LIN {X 0,Y 573.233,Z 312.707,A -85,B 0,C 180,E1 -2302.192,E2 -2302.192} C_VEL
LIN {X 0,Y 573.235,Z 312.7,A -85,B 0,C 180,E1 -2305.229,E2 -2305.229} C_VEL
LIN {X 0,Y 573.253,Z 312.699,A -85,B 0,C 180,E1 -2307.772,E2 -2307.772} C_VEL
LIN {X 0,Y 573.264,Z 312.7,A -85,B 0,C 180,E1 -2310.634,E2 -2310.634} C_VEL
LIN {X 0,Y 573.212,Z 312.703,A -85,B 0,C 180,E1 -2313.514,E2 -2313.514} C_VEL
LIN {X 0,Y 573.23,Z 312.71,A -85,B 0,C 180,E1 -2316.135,E2 -2316.135} C_VEL
LIN {X 0,Y 573.252,Z 312.697,A -85,B 0,C 180,E1 -2319.174,E2 -2319.174} C_VEL
LIN {X 0,Y 573.218,Z 312.702,A -85,B 0,C 180,E1 -2321.411,E2 -2321.411} C_VEL
LIN {X 0,Y 573.244,Z 312.701,A -85,B 0,C 180,E1 -2323.622,E2 -2323.622} C_VEL
LIN {X 0,Y 573.276,Z 312.7,A -85,B 0,C 180,E1 -2325.807,E2 -2325.807} C_VEL
LIN {X 0,Y 573.268,Z 312.696,A -85,B 0,C 180,E1 -2328.745,E2 -2328.745} C_VEL
LIN {X 0,Y 573.254,Z 312.7,A -85,B 0,C 180,E1 -2331.54,E2 -2331.54} C_VEL
LIN {X 0,Y 573.274,Z 312.698,A -85,B 0,C 180,E1 -2334.372,E2 -2334.372} C_VEL
LIN {X 0,Y 573.308,Z 312.699,A -85,B 0,C 180,E1 -2337.893,E2 -2337.893} C_VEL
LIN {X 0,Y 573.318,Z 312.697,A -85,B 0,C 180,E1 -2340,E2 -2340} C_VEL
LIN {X 0,Y 573.287,Z 312.693,A -85,B 0,C 180,E1 -2342.811,E2 -2342.811} C_VEL
LIN {X 0,Y 573.28,Z 312.701,A -85,B 0,C 180,E1 -2345.629,E2 -2345.629} C_VEL
LIN {X 0,Y 573.239,Z 312.7,A -85,B 0,C 180,E1 -2348.46,E2 -2348.46} C_VEL
LIN {X 0,Y 573.277,Z 312.697,A -85,B 0,C 180,E1 -2351.312,E2 -2351.312} C_VEL
LIN {X 0,Y 573.262,Z 312.697,A -85,B 0,C 180,E1 -2354.415,E2 -2354.415} C_VEL
LIN {X 0,Y 573.181,Z 312.707,A -85,B 0,C 180,E1 -2357.114,E2 -2357.114} C_VEL
LIN {X 0,Y 573.27,Z 312.7,A -85,B 0,C 180,E1 -2359.33,E2 -2359.33} C_VEL
LIN {X 0,Y 573.199,Z 312.705,A -85,B 0,C 180,E1 -2362.34,E2 -2362.34} C_VEL
LIN {X 0,Y 573.197,Z 312.704,A -85,B 0,C 180,E1 -2364.342,E2 -2364.342} C_VEL
LIN {X 0,Y 572.56,Z 312.785,A -85,B 0,C 180,E1 -2364.928,E2 -2364.928} C_VEL
LIN {X 0,Y 569.728,Z 313.143,A -85,B 0,C 180,E1 -2365.88,E2 -2365.88} C_VEL
LIN {X 0,Y 567.308,Z 313.449,A -85,B 0,C 180,E1 -2366.645,E2 -2366.645} C_VEL
LIN {X 0,Y 566.25,Z 313.578,A -85,B 0,C 180,E1 -2367.236,E2 -2367.236} C_VEL
LIN {X 0,Y 566.155,Z 313.587,A -85,B 0,C 180,E1 -2367.437,E2 -2367.437} C_VEL
LIN {X 0,Y 566.151,Z 313.584,A -85,B 0,C 180,E1 -2369.772,E2 -2369.772} C_VEL
LIN {X 0,Y 566.181,Z 313.578,A -85,B 0,C 180,E1 -2372.425,E2 -2372.425} C_VEL
LIN {X 0,Y 566.162,Z 313.584,A -85,B 0,C 180,E1 -2374.986,E2 -2374.986} C_VEL
LIN {X 0,Y 566.18,Z 313.586,A -85,B 0,C 180,E1 -2377.463,E2 -2377.463} C_VEL
LIN {X 0,Y 566.159,Z 313.581,A -85,B 0,C 180,E1 -2380.204,E2 -2380.204} C_VEL
LIN {X 0,Y 566.145,Z 313.589,A -85,B 0,C 180,E1 -2383.06,E2 -2383.06} C_VEL
LIN {X 0,Y 566.136,Z 313.584,A -85,B 0,C 180,E1 -2386.056,E2 -2386.056} C_VEL
LIN {X 0,Y 566.124,Z 313.59,A -85,B 0,C 180,E1 -2388.856,E2 -2388.856} C_VEL
LIN {X 0,Y 566.157,Z 313.589,A -85,B 0,C 180,E1 -2391.449,E2 -2391.449} C_VEL
LIN {X 0,Y 566.135,Z 313.585,A -85,B 0,C 180,E1 -2394.306,E2 -2394.306} C_VEL
LIN {X 0,Y 566.154,Z 313.588,A -85,B 0,C 180,E1 -2396.893,E2 -2396.893} C_VEL
LIN {X 0,Y 566.151,Z 313.59,A -85,B 0,C 180,E1 -2399.405,E2 -2399.405} C_VEL
LIN {X 0,Y 566.145,Z 313.587,A -85,B 0,C 180,E1 -2401.854,E2 -2401.854} C_VEL
LIN {X 0,Y 566.187,Z 313.691,A -85,B 0,C 180,E1 -2403.507,E2 -2403.507} C_VEL
LIN {X 0,Y 566.832,Z 319.406,A -85,B 0,C 180,E1 -2404.447,E2 -2404.447} C_VEL
LIN {X 0,Y 566.58,Z 337.004,A -85,B 0,C 180,E1 -2407.193,E2 -2407.193} C_VEL
LIN {X 0,Y 566.557,Z 342.716,A -85,B 0,C 180,E1 -2408.077,E2 -2408.077} C_VEL
LIN {X 0,Y 567.74,Z 348.996,A -85,B 0,C 180,E1 -2408.2,E2 -2408.2} C_VEL
LIN {X 0,Y 567.437,Z 479.381,A -85,B 0,C 180,E1 -2409.89,E2 -2409.89} C_VEL
LIN {X 0,Y 567.328,Z 493.858,A -85,B 0,C 180,E1 -2410.226,E2 -2410.226} C_VEL
LIN {X 0,Y 567.16,Z 507.522,A -85,B 0,C 180,E1 -2410.689,E2 -2410.689} C_VEL
LIN {X 0,Y 567.009,Z 520.891,A -85,B 0,C 180,E1 -2411.294,E2 -2411.294} C_VEL
LIN {X 0,Y 566.777,Z 533.749,A -85,B 0,C 180,E1 -2412.034,E2 -2412.034} C_VEL
LIN {X 0,Y 566.592,Z 545.641,A -85,B 0,C 180,E1 -2412.884,E2 -2412.884} C_VEL
LIN {X 0,Y 566.402,Z 556.077,A -85,B 0,C 180,E1 -2413.788,E2 -2413.788} C_VEL
LIN {X 0,Y 566.259,Z 566.633,A -85,B 0,C 180,E1 -2414.892,E2 -2414.892} C_VEL
LIN {X 0,Y 566.111,Z 575.295,A -85,B 0,C 180,E1 -2415.99,E2 -2415.99} C_VEL
LIN {X 0,Y 566.022,Z 583.527,A -85,B 0,C 180,E1 -2417.268,E2 -2417.268} C_VEL
LIN {X 0,Y 565.938,Z 590.127,A -85,B 0,C 180,E1 -2418.539,E2 -2418.539} C_VEL
LIN {X 0,Y 565.917,Z 594.689,A -85,B 0,C 180,E1 -2419.626,E2 -2419.626} C_VEL
LIN {X 0,Y 565.877,Z 598.259,A -85,B 0,C 180,E1 -2420.709,E2 -2420.709} C_VEL
LIN {X 0,Y 565.882,Z 601.734,A -85,B 0,C 180,E1 -2422.148,E2 -2422.148} C_VEL
LIN {X 0,Y 565.899,Z 603.791,A -85,B 0,C 180,E1 -2423.582,E2 -2423.582} C_VEL
LIN {X 0,Y 565.843,Z 604.498,A -85,B 0,C 180,E1 -2425.012,E2 -2425.012} C_VEL
LIN {X 0,Y 565.885,Z 603.864,A -85,B 0,C 180,E1 -2426.44,E2 -2426.44} C_VEL
LIN {X 0,Y 565.839,Z 601.889,A -85,B 0,C 180,E1 -2427.865,E2 -2427.865} C_VEL
LIN {X 0,Y 565.848,Z 598.534,A -85,B 0,C 180,E1 -2429.288,E2 -2429.288} C_VEL
LIN {X 0,Y 565.89,Z 593.71,A -85,B 0,C 180,E1 -2430.712,E2 -2430.712} C_VEL
LIN {X 0,Y 566.002,Z 589.069,A -85,B 0,C 180,E1 -2431.779,E2 -2431.779} C_VEL
LIN {X 0,Y 566.061,Z 582.343,A -85,B 0,C 180,E1 -2433.025,E2 -2433.025} C_VEL
LIN {X 0,Y 566.16,Z 574.011,A -85,B 0,C 180,E1 -2434.271,E2 -2434.271} C_VEL
LIN {X 0,Y 566.241,Z 565.352,A -85,B 0,C 180,E1 -2435.341,E2 -2435.341} C_VEL
LIN {X 0,Y 566.433,Z 554.892,A -85,B 0,C 180,E1 -2436.411,E2 -2436.411} C_VEL
LIN {X 0,Y 566.652,Z 543.21,A -85,B 0,C 180,E1 -2437.393,E2 -2437.393} C_VEL
LIN {X 0,Y 566.792,Z 531.518,A -85,B 0,C 180,E1 -2438.198,E2 -2438.198} C_VEL
LIN {X 0,Y 566.976,Z 518.644,A -85,B 0,C 180,E1 -2438.914,E2 -2438.914} C_VEL
LIN {X 0,Y 567.241,Z 505.16,A -85,B 0,C 180,E1 -2439.494,E2 -2439.494} C_VEL
LIN {X 0,Y 567.35,Z 491.016,A -85,B 0,C 180,E1 -2439.942,E2 -2439.942} C_VEL
LIN {X 0,Y 567.445,Z 477.281,A -85,B 0,C 180,E1 -2440.233,E2 -2440.233} C_VEL
LIN {X 0,Y 567.725,Z 349.043,A -85,B 0,C 180,E1 -2441.89,E2 -2441.89} C_VEL
LIN {X 0,Y 566.529,Z 342.625,A -85,B 0,C 180,E1 -2442.028,E2 -2442.028} C_VEL
LIN {X 0,Y 566.725,Z 325.458,A -85,B 0,C 180,E1 -2444.694,E2 -2444.694} C_VEL
LIN {X 0,Y 566.648,Z 315.932,A -85,B 0,C 180,E1 -2446.204,E2 -2446.204} C_VEL
LIN {X 0,Y 566.21,Z 313.584,A -85,B 0,C 180,E1 -2446.62,E2 -2446.62} C_VEL
LIN {X 0,Y 566.174,Z 313.583,A -85,B 0,C 180,E1 -2449.582,E2 -2449.582} C_VEL
LIN {X 0,Y 566.153,Z 313.583,A -85,B 0,C 180,E1 -2451.864,E2 -2451.864} C_VEL
LIN {X 0,Y 566.148,Z 313.584,A -85,B 0,C 180,E1 -2454.183,E2 -2454.183} C_VEL
LIN {X 0,Y 566.16,Z 313.588,A -85,B 0,C 180,E1 -2456.648,E2 -2456.648} C_VEL
LIN {X 0,Y 566.137,Z 313.584,A -85,B 0,C 180,E1 -2459.659,E2 -2459.659} C_VEL
LIN {X 0,Y 566.171,Z 313.584,A -85,B 0,C 180,E1 -2462.424,E2 -2462.424} C_VEL
LIN {X 0,Y 566.158,Z 313.588,A -85,B 0,C 180,E1 -2464.985,E2 -2464.985} C_VEL
LIN {X 0,Y 566.158,Z 313.582,A -85,B 0,C 180,E1 -2467.464,E2 -2467.464} C_VEL
LIN {X 0,Y 566.165,Z 313.583,A -85,B 0,C 180,E1 -2470.203,E2 -2470.203} C_VEL
LIN {X 0,Y 566.139,Z 313.588,A -85,B 0,C 180,E1 -2473.06,E2 -2473.06} C_VEL
LIN {X 0,Y 566.147,Z 313.584,A -85,B 0,C 180,E1 -2476.055,E2 -2476.055} C_VEL
LIN {X 0,Y 566.141,Z 313.589,A -85,B 0,C 180,E1 -2478.857,E2 -2478.857} C_VEL
LIN {X 0,Y 566.159,Z 313.581,A -85,B 0,C 180,E1 -2481.449,E2 -2481.449} C_VEL
LIN {X 0,Y 566.161,Z 313.581,A -85,B 0,C 180,E1 -2483.792,E2 -2483.792} C_VEL
LIN {X 0,Y 566.199,Z 313.582,A -85,B 0,C 180,E1 -2486.269,E2 -2486.269} C_VEL
LIN {X 0,Y 566.179,Z 313.582,A -85,B 0,C 180,E1 -2488.926,E2 -2488.926} C_VEL
LIN {X 0,Y 566.145,Z 313.584,A -85,B 0,C 180,E1 -2491.853,E2 -2491.853} C_VEL
LIN {X 0,Y 566.192,Z 313.583,A -85,B 0,C 180,E1 -2494.25,E2 -2494.25} C_VEL
LIN {X 0,Y 566.151,Z 313.586,A -85,B 0,C 180,E1 -2496.724,E2 -2496.724} C_VEL
LIN {X 0,Y 566.194,Z 313.575,A -85,B 0,C 180,E1 -2498.901,E2 -2498.901} C_VEL
LIN {X 0,Y 566.187,Z 313.576,A -85,B 0,C 180,E1 -2501.171,E2 -2501.171} C_VEL
LIN {X 0,Y 566.175,Z 313.587,A -85,B 0,C 180,E1 -2504.152,E2 -2504.152} C_VEL
LIN {X 0,Y 566.169,Z 313.586,A -85,B 0,C 180,E1 -2506.358,E2 -2506.358} C_VEL
LIN {X 0,Y 566.234,Z 313.567,A -85,B 0,C 180,E1 -2509.27,E2 -2509.27} C_VEL
LIN {X 0,Y 566.22,Z 313.582,A -85,B 0,C 180,E1 -2512.152,E2 -2512.152} C_VEL
LIN {X 0,Y 566.261,Z 313.568,A -85,B 0,C 180,E1 -2515.016,E2 -2515.016} C_VEL
LIN {X 0,Y 566.277,Z 313.572,A -85,B 0,C 180,E1 -2517.866,E2 -2517.866} C_VEL
LIN {X 0,Y 566.299,Z 313.564,A -85,B 0,C 180,E1 -2520.711,E2 -2520.711} C_VEL
LIN {X 0,Y 566.259,Z 313.569,A -85,B 0,C 180,E1 -2522.845,E2 -2522.845} C_VEL
LIN {X 0,Y 566.244,Z 313.575,A -85,B 0,C 180,E1 -2525.698,E2 -2525.698} C_VEL
LIN {X 0,Y 566.205,Z 313.577,A -85,B 0,C 180,E1 -2528.566,E2 -2528.566} C_VEL
LIN {X 0,Y 566.246,Z 313.573,A -85,B 0,C 180,E1 -2531.454,E2 -2531.454} C_VEL
LIN {X 0,Y 566.238,Z 313.573,A -85,B 0,C 180,E1 -2534.506,E2 -2534.506} C_VEL
LIN {X 0,Y 566.197,Z 313.579,A -85,B 0,C 180,E1 -2537.332,E2 -2537.332} C_VEL
LIN {X 0,Y 566.208,Z 313.578,A -85,B 0,C 180,E1 -2540.337,E2 -2540.337} C_VEL
LIN {X 0,Y 566.171,Z 313.582,A -85,B 0,C 180,E1 -2543.28,E2 -2543.28} C_VEL
LIN {X 0,Y 566.211,Z 313.584,A -85,B 0,C 180,E1 -2545.749,E2 -2545.749} C_VEL
LIN {X 0,Y 566.186,Z 313.578,A -85,B 0,C 180,E1 -2548.954,E2 -2548.954} C_VEL
LIN {X 0,Y 566.195,Z 313.583,A -85,B 0,C 180,E1 -2551.422,E2 -2551.422} C_VEL
LIN {X 0,Y 566.212,Z 313.581,A -85,B 0,C 180,E1 -2553.956,E2 -2553.956} C_VEL
LIN {X 0,Y 566.191,Z 313.578,A -85,B 0,C 180,E1 -2556.571,E2 -2556.571} C_VEL
LIN {X 0,Y 566.215,Z 313.583,A -85,B 0,C 180,E1 -2559.685,E2 -2559.685} C_VEL
LIN {X 0,Y 566.203,Z 313.578,A -85,B 0,C 180,E1 -2562.917,E2 -2562.917} C_VEL
LIN {X 0,Y 566.195,Z 313.579,A -85,B 0,C 180,E1 -2566.049,E2 -2566.049} C_VEL
LIN {X 0,Y 566.205,Z 313.581,A -85,B 0,C 180,E1 -2569.214,E2 -2569.214} C_VEL
LIN {X 0,Y 566.187,Z 313.586,A -85,B 0,C 180,E1 -2571.637,E2 -2571.637} C_VEL
LIN {X 0,Y 566.198,Z 313.578,A -85,B 0,C 180,E1 -2574.31,E2 -2574.31} C_VEL
LIN {X 0,Y 566.222,Z 313.577,A -85,B 0,C 180,E1 -2576.898,E2 -2576.898} C_VEL
LIN {X 0,Y 566.182,Z 313.588,A -85,B 0,C 180,E1 -2579.407,E2 -2579.407} C_VEL
LIN {X 0,Y 566.214,Z 313.578,A -85,B 0,C 180,E1 -2581.857,E2 -2581.857} C_VEL
LIN {X 0,Y 566.215,Z 313.577,A -85,B 0,C 180,E1 -2584.251,E2 -2584.251} C_VEL
LIN {X 0,Y 566.257,Z 313.606,A -85,B 0,C 180,E1 -2585.236,E2 -2585.236} C_VEL
LIN {X 0,Y 567.337,Z 319.181,A -85,B 0,C 180,E1 -2586.042,E2 -2586.042} C_VEL
LIN {X 0,Y 567.184,Z 336.227,A -85,B 0,C 180,E1 -2588.33,E2 -2588.33} C_VEL
LIN {X 0,Y 566.852,Z 359.12,A -85,B 0,C 180,E1 -2591.382,E2 -2591.382} C_VEL
LIN {X 0,Y 566.677,Z 371.554,A -85,B 0,C 180,E1 -2593.018,E2 -2593.018} C_VEL
LIN {X 0,Y 567.808,Z 378.423,A -85,B 0,C 180,E1 -2593.15,E2 -2593.15} C_VEL
LIN {X 0,Y 567.462,Z 508.628,A -85,B 0,C 180,E1 -2594.833,E2 -2594.833} C_VEL
LIN {X 0,Y 567.304,Z 523.138,A -85,B 0,C 180,E1 -2595.159,E2 -2595.159} C_VEL
LIN {X 0,Y 567.204,Z 536.383,A -85,B 0,C 180,E1 -2595.598,E2 -2595.598} C_VEL
LIN {X 0,Y 566.995,Z 549.875,A -85,B 0,C 180,E1 -2596.196,E2 -2596.196} C_VEL
LIN {X 0,Y 566.771,Z 562.678,A -85,B 0,C 180,E1 -2596.921,E2 -2596.921} C_VEL
LIN {X 0,Y 566.617,Z 574.312,A -85,B 0,C 180,E1 -2597.736,E2 -2597.736} C_VEL
LIN {X 0,Y 566.444,Z 584.221,A -85,B 0,C 180,E1 -2598.571,E2 -2598.571} C_VEL
LIN {X 0,Y 566.294,Z 594.706,A -85,B 0,C 180,E1 -2599.633,E2 -2599.633} C_VEL
LIN {X 0,Y 566.177,Z 603.558,A -85,B 0,C 180,E1 -2600.714,E2 -2600.714} C_VEL
LIN {X 0,Y 566.047,Z 612.036,A -85,B 0,C 180,E1 -2601.971,E2 -2601.971} C_VEL
LIN {X 0,Y 565.966,Z 619.802,A -85,B 0,C 180,E1 -2603.422,E2 -2603.422} C_VEL
LIN {X 0,Y 565.928,Z 624.961,A -85,B 0,C 180,E1 -2604.656,E2 -2604.656} C_VEL
LIN {X 0,Y 565.956,Z 628.443,A -85,B 0,C 180,E1 -2605.727,E2 -2605.727} C_VEL
LIN {X 0,Y 565.874,Z 631.832,A -85,B 0,C 180,E1 -2607.152,E2 -2607.152} C_VEL
LIN {X 0,Y 565.84,Z 633.833,A -85,B 0,C 180,E1 -2608.577,E2 -2608.577} C_VEL
LIN {X 0,Y 565.837,Z 634.5,A -85,B 0,C 180,E1 -2610,E2 -2610} C_VEL
LIN {X 0,Y 565.84,Z 633.834,A -85,B 0,C 180,E1 -2611.423,E2 -2611.423} C_VEL
LIN {X 0,Y 565.874,Z 631.834,A -85,B 0,C 180,E1 -2612.848,E2 -2612.848} C_VEL
LIN {X 0,Y 565.956,Z 628.445,A -85,B 0,C 180,E1 -2614.273,E2 -2614.273} C_VEL
LIN {X 0,Y 565.988,Z 623.568,A -85,B 0,C 180,E1 -2615.701,E2 -2615.701} C_VEL
LIN {X 0,Y 565.993,Z 619.044,A -85,B 0,C 180,E1 -2616.739,E2 -2616.739} C_VEL
LIN {X 0,Y 566.047,Z 612.036,A -85,B 0,C 180,E1 -2618.029,E2 -2618.029} C_VEL
LIN {X 0,Y 566.177,Z 603.557,A -85,B 0,C 180,E1 -2619.287,E2 -2619.287} C_VEL
LIN {X 0,Y 566.294,Z 594.706,A -85,B 0,C 180,E1 -2620.367,E2 -2620.367} C_VEL
LIN {X 0,Y 566.485,Z 583.988,A -85,B 0,C 180,E1 -2621.449,E2 -2621.449} C_VEL
LIN {X 0,Y 566.608,Z 573.138,A -85,B 0,C 180,E1 -2622.355,E2 -2622.355} C_VEL
LIN {X 0,Y 566.78,Z 561.253,A -85,B 0,C 180,E1 -2623.171,E2 -2623.171} C_VEL
LIN {X 0,Y 567.023,Z 548.093,A -85,B 0,C 180,E1 -2623.895,E2 -2623.895} C_VEL
LIN {X 0,Y 567.198,Z 535.022,A -85,B 0,C 180,E1 -2624.455,E2 -2624.455} C_VEL
LIN {X 0,Y 567.338,Z 520.511,A -85,B 0,C 180,E1 -2624.91,E2 -2624.91} C_VEL
LIN {X 0,Y 567.452,Z 507.12,A -85,B 0,C 180,E1 -2625.19,E2 -2625.19} C_VEL
LIN {X 0,Y 567.684,Z 377.239,A -85,B 0,C 180,E1 -2626.87,E2 -2626.87} C_VEL
LIN {X 0,Y 566.669,Z 371.553,A -85,B 0,C 180,E1 -2626.982,E2 -2626.982} C_VEL
LIN {X 0,Y 566.953,Z 351.768,A -85,B 0,C 180,E1 -2629.592,E2 -2629.592} C_VEL
LIN {X 0,Y 567.279,Z 330.788,A -85,B 0,C 180,E1 -2632.393,E2 -2632.393} C_VEL
LIN {X 0,Y 567.32,Z 319.163,A -85,B 0,C 180,E1 -2633.958,E2 -2633.958} C_VEL
LIN {X 0,Y 566.241,Z 313.581,A -85,B 0,C 180,E1 -2634.789,E2 -2634.789} C_VEL
LIN {X 0,Y 566.21,Z 313.578,A -85,B 0,C 180,E1 -2637.339,E2 -2637.339} C_VEL
LIN {X 0,Y 566.204,Z 313.576,A -85,B 0,C 180,E1 -2639.769,E2 -2639.769} C_VEL
LIN {X 0,Y 566.206,Z 313.583,A -85,B 0,C 180,E1 -2642.43,E2 -2642.43} C_VEL
LIN {X 0,Y 566.184,Z 313.583,A -85,B 0,C 180,E1 -2644.99,E2 -2644.99} C_VEL
LIN {X 0,Y 566.198,Z 313.577,A -85,B 0,C 180,E1 -2647.461,E2 -2647.461} C_VEL
LIN {X 0,Y 566.209,Z 313.58,A -85,B 0,C 180,E1 -2650.199,E2 -2650.199} C_VEL
LIN {X 0,Y 566.202,Z 313.577,A -85,B 0,C 180,E1 -2653.055,E2 -2653.055} C_VEL
LIN {X 0,Y 566.196,Z 313.58,A -85,B 0,C 180,E1 -2656.05,E2 -2656.05} C_VEL
LIN {X 0,Y 566.206,Z 313.576,A -85,B 0,C 180,E1 -2659.215,E2 -2659.215} C_VEL
LIN {X 0,Y 566.184,Z 313.578,A -85,B 0,C 180,E1 -2661.637,E2 -2661.637} C_VEL
LIN {X 0,Y 566.153,Z 313.591,A -85,B 0,C 180,E1 -2664.307,E2 -2664.307} C_VEL
LIN {X 0,Y 566.223,Z 313.575,A -85,B 0,C 180,E1 -2666.898,E2 -2666.898} C_VEL
LIN {X 0,Y 566.182,Z 313.578,A -85,B 0,C 180,E1 -2669.407,E2 -2669.407} C_VEL
LIN {X 0,Y 566.19,Z 313.581,A -85,B 0,C 180,E1 -2671.856,E2 -2671.856} C_VEL
LIN {X 0,Y 566.241,Z 313.571,A -85,B 0,C 180,E1 -2675.039,E2 -2675.039} C_VEL
LIN {X 0,Y 566.196,Z 313.585,A -85,B 0,C 180,E1 -2678.138,E2 -2678.138} C_VEL
LIN {X 0,Y 566.235,Z 313.574,A -85,B 0,C 180,E1 -2680.614,E2 -2680.614} C_VEL
LIN {X 0,Y 566.212,Z 313.575,A -85,B 0,C 180,E1 -2683.412,E2 -2683.412} C_VEL
LIN {X 0,Y 566.192,Z 313.581,A -85,B 0,C 180,E1 -2686.359,E2 -2686.359} C_VEL
LIN {X 0,Y 566.238,Z 313.572,A -85,B 0,C 180,E1 -2689.27,E2 -2689.27} C_VEL
LIN {X 0,Y 566.196,Z 313.583,A -85,B 0,C 180,E1 -2692.153,E2 -2692.153} C_VEL
LIN {X 0,Y 566.271,Z 313.567,A -85,B 0,C 180,E1 -2695.016,E2 -2695.016} C_VEL
LIN {X 0,Y 566.279,Z 313.574,A -85,B 0,C 180,E1 -2697.866,E2 -2697.866} C_VEL
LIN {X 0,Y 566.287,Z 313.573,A -85,B 0,C 180,E1 -2700,E2 -2700} C_VEL
LIN {X 0,Y 566.256,Z 313.569,A -85,B 0,C 180,E1 -2702.846,E2 -2702.846} C_VEL
LIN {X 0,Y 566.247,Z 313.578,A -85,B 0,C 180,E1 -2705.699,E2 -2705.699} C_VEL
LIN {X 0,Y 566.193,Z 313.577,A -85,B 0,C 180,E1 -2708.566,E2 -2708.566} C_VEL
LIN {X 0,Y 566.244,Z 313.575,A -85,B 0,C 180,E1 -2711.455,E2 -2711.455} C_VEL
LIN {X 0,Y 566.218,Z 313.574,A -85,B 0,C 180,E1 -2714.498,E2 -2714.498} C_VEL
LIN {X 0,Y 566.155,Z 313.585,A -85,B 0,C 180,E1 -2717.333,E2 -2717.333} C_VEL
LIN {X 0,Y 566.195,Z 313.586,A -85,B 0,C 180,E1 -2719.581,E2 -2719.581} C_VEL
LIN {X 0,Y 566.151,Z 313.588,A -85,B 0,C 180,E1 -2721.865,E2 -2721.865} C_VEL
LIN {X 0,Y 566.183,Z 313.579,A -85,B 0,C 180,E1 -2725.021,E2 -2725.021} C_VEL
LIN {X 0,Y 566.155,Z 313.587,A -85,B 0,C 180,E1 -2727.437,E2 -2727.437} C_VEL
LIN {X 0,Y 565.459,Z 313.67,A -85,B 0,C 180,E1 -2728.031,E2 -2728.031} C_VEL
LIN {X 0,Y 562.585,Z 314.028,A -85,B 0,C 180,E1 -2728.994,E2 -2728.994} C_VEL
LIN {X 0,Y 560.185,Z 314.326,A -85,B 0,C 180,E1 -2729.77,E2 -2729.77} C_VEL
LIN {X 0,Y 559.174,Z 314.447,A -85,B 0,C 180,E1 -2730.369,E2 -2730.369} C_VEL
LIN {X 0,Y 559.101,Z 314.456,A -85,B 0,C 180,E1 -2730.572,E2 -2730.572} C_VEL
LIN {X 0,Y 559.139,Z 314.456,A -85,B 0,C 180,E1 -2732.717,E2 -2732.717} C_VEL
LIN {X 0,Y 559.115,Z 314.467,A -85,B 0,C 180,E1 -2735.325,E2 -2735.325} C_VEL
LIN {X 0,Y 559.1,Z 314.462,A -85,B 0,C 180,E1 -2738.021,E2 -2738.021} C_VEL
LIN {X 0,Y 559.095,Z 314.463,A -85,B 0,C 180,E1 -2740.818,E2 -2740.818} C_VEL
LIN {X 0,Y 559.095,Z 314.465,A -85,B 0,C 180,E1 -2743.739,E2 -2743.739} C_VEL
LIN {X 0,Y 559.086,Z 314.462,A -85,B 0,C 180,E1 -2746.26,E2 -2746.26} C_VEL
LIN {X 0,Y 559.087,Z 314.471,A -85,B 0,C 180,E1 -2749.181,E2 -2749.181} C_VEL
LIN {X 0,Y 559.116,Z 314.469,A -85,B 0,C 180,E1 -2751.2,E2 -2751.2} C_VEL
LIN {X 0,Y 559.111,Z 314.462,A -85,B 0,C 180,E1 -2753.787,E2 -2753.787} C_VEL
LIN {X 0,Y 559.113,Z 314.46,A -85,B 0,C 180,E1 -2756.421,E2 -2756.421} C_VEL
LIN {X 0,Y 559.137,Z 314.464,A -85,B 0,C 180,E1 -2758.979,E2 -2758.979} C_VEL
LIN {X 0,Y 559.107,Z 314.466,A -85,B 0,C 180,E1 -2761.632,E2 -2761.632} C_VEL
LIN {X 0,Y 559.173,Z 314.585,A -85,B 0,C 180,E1 -2763.344,E2 -2763.344} C_VEL
LIN {X 0,Y 559.866,Z 319.282,A -85,B 0,C 180,E1 -2764.137,E2 -2764.137} C_VEL
LIN {X 0,Y 559.637,Z 336.767,A -85,B 0,C 180,E1 -2766.926,E2 -2766.926} C_VEL
LIN {X 0,Y 559.549,Z 342.783,A -85,B 0,C 180,E1 -2767.864,E2 -2767.864} C_VEL
LIN {X 0,Y 560.977,Z 350.661,A -85,B 0,C 180,E1 -2768.012,E2 -2768.012} C_VEL
LIN {X 0,Y 560.59,Z 479.985,A -85,B 0,C 180,E1 -2769.713,E2 -2769.713} C_VEL
LIN {X 0,Y 560.47,Z 494.26,A -85,B 0,C 180,E1 -2770.053,E2 -2770.053} C_VEL
LIN {X 0,Y 560.239,Z 508.368,A -85,B 0,C 180,E1 -2770.542,E2 -2770.542} C_VEL
LIN {X 0,Y 560.082,Z 521.43,A -85,B 0,C 180,E1 -2771.148,E2 -2771.148} C_VEL
LIN {X 0,Y 559.831,Z 534.183,A -85,B 0,C 180,E1 -2771.898,E2 -2771.898} C_VEL
LIN {X 0,Y 559.609,Z 546.039,A -85,B 0,C 180,E1 -2772.762,E2 -2772.762} C_VEL
LIN {X 0,Y 559.376,Z 557.352,A -85,B 0,C 180,E1 -2773.767,E2 -2773.767} C_VEL
LIN {X 0,Y 559.211,Z 567.779,A -85,B 0,C 180,E1 -2774.902,E2 -2774.902} C_VEL
LIN {X 0,Y 559.068,Z 576.126,A -85,B 0,C 180,E1 -2775.997,E2 -2775.997} C_VEL
LIN {X 0,Y 558.955,Z 584.194,A -85,B 0,C 180,E1 -2777.289,E2 -2777.289} C_VEL
LIN {X 0,Y 558.861,Z 589.841,A -85,B 0,C 180,E1 -2778.392,E2 -2778.392} C_VEL
LIN {X 0,Y 558.843,Z 594.441,A -85,B 0,C 180,E1 -2779.493,E2 -2779.493} C_VEL
LIN {X 0,Y 558.794,Z 598.071,A -85,B 0,C 180,E1 -2780.59,E2 -2780.59} C_VEL
LIN {X 0,Y 558.802,Z 601.609,A -85,B 0,C 180,E1 -2782.048,E2 -2782.048} C_VEL
LIN {X 0,Y 558.828,Z 603.723,A -85,B 0,C 180,E1 -2783.501,E2 -2783.501} C_VEL
LIN {X 0,Y 558.758,Z 604.485,A -85,B 0,C 180,E1 -2784.949,E2 -2784.949} C_VEL
LIN {X 0,Y 558.797,Z 603.919,A -85,B 0,C 180,E1 -2786.395,E2 -2786.395} C_VEL
LIN {X 0,Y 558.745,Z 602.012,A -85,B 0,C 180,E1 -2787.837,E2 -2787.837} C_VEL
LIN {X 0,Y 558.75,Z 598.719,A -85,B 0,C 180,E1 -2789.279,E2 -2789.279} C_VEL
LIN {X 0,Y 558.796,Z 593.958,A -85,B 0,C 180,E1 -2790.721,E2 -2790.721} C_VEL
LIN {X 0,Y 558.911,Z 589.374,A -85,B 0,C 180,E1 -2791.801,E2 -2791.801} C_VEL
LIN {X 0,Y 559.008,Z 582.725,A -85,B 0,C 180,E1 -2793.063,E2 -2793.063} C_VEL
LIN {X 0,Y 559.12,Z 574.48,A -85,B 0,C 180,E1 -2794.325,E2 -2794.325} C_VEL
LIN {X 0,Y 559.21,Z 565.917,A -85,B 0,C 180,E1 -2795.409,E2 -2795.409} C_VEL
LIN {X 0,Y 559.411,Z 555.568,A -85,B 0,C 180,E1 -2796.492,E2 -2796.492} C_VEL
LIN {X 0,Y 559.659,Z 544.021,A -85,B 0,C 180,E1 -2797.486,E2 -2797.486} C_VEL
LIN {X 0,Y 559.842,Z 532.5,A -85,B 0,C 180,E1 -2798.301,E2 -2798.301} C_VEL
LIN {X 0,Y 560.041,Z 519.861,A -85,B 0,C 180,E1 -2799.025,E2 -2799.025} C_VEL
LIN {X 0,Y 560.319,Z 506.76,A -85,B 0,C 180,E1 -2799.612,E2 -2799.612} C_VEL
LIN {X 0,Y 560.49,Z 492.577,A -85,B 0,C 180,E1 -2800.088,E2 -2800.088} C_VEL
LIN {X 0,Y 560.602,Z 478.446,A -85,B 0,C 180,E1 -2800.405,E2 -2800.405} C_VEL
LIN {X 0,Y 560.878,Z 349.648,A -85,B 0,C 180,E1 -2802.094,E2 -2802.094} C_VEL
LIN {X 0,Y 559.518,Z 342.657,A -85,B 0,C 180,E1 -2802.243,E2 -2802.243} C_VEL
LIN {X 0,Y 559.771,Z 326.369,A -85,B 0,C 180,E1 -2804.816,E2 -2804.816} C_VEL
LIN {X 0,Y 559.763,Z 317.67,A -85,B 0,C 180,E1 -2806.222,E2 -2806.222} C_VEL
LIN {X 0,Y 559.17,Z 314.462,A -85,B 0,C 180,E1 -2806.803,E2 -2806.803} C_VEL
LIN {X 0,Y 559.138,Z 314.458,A -85,B 0,C 180,E1 -2809.839,E2 -2809.839} C_VEL
LIN {X 0,Y 559.11,Z 314.461,A -85,B 0,C 180,E1 -2812.154,E2 -2812.154} C_VEL
LIN {X 0,Y 559.087,Z 314.467,A -85,B 0,C 180,E1 -2814.509,E2 -2814.509} C_VEL
LIN {X 0,Y 559.11,Z 314.47,A -85,B 0,C 180,E1 -2816.906,E2 -2816.906} C_VEL
LIN {X 0,Y 559.087,Z 314.462,A -85,B 0,C 180,E1 -2819.845,E2 -2819.845} C_VEL
LIN {X 0,Y 559.128,Z 314.466,A -85,B 0,C 180,E1 -2822.717,E2 -2822.717} C_VEL
LIN {X 0,Y 559.113,Z 314.461,A -85,B 0,C 180,E1 -2825.325,E2 -2825.325} C_VEL
LIN {X 0,Y 559.093,Z 314.462,A -85,B 0,C 180,E1 -2828.021,E2 -2828.021} C_VEL
LIN {X 0,Y 559.1,Z 314.468,A -85,B 0,C 180,E1 -2830.818,E2 -2830.818} C_VEL
LIN {X 0,Y 559.087,Z 314.462,A -85,B 0,C 180,E1 -2833.74,E2 -2833.74} C_VEL
LIN {X 0,Y 559.095,Z 314.465,A -85,B 0,C 180,E1 -2836.261,E2 -2836.261} C_VEL
LIN {X 0,Y 559.096,Z 314.463,A -85,B 0,C 180,E1 -2839.182,E2 -2839.182} C_VEL
LIN {X 0,Y 559.1,Z 314.462,A -85,B 0,C 180,E1 -2841.979,E2 -2841.979} C_VEL
LIN {X 0,Y 559.123,Z 314.463,A -85,B 0,C 180,E1 -2844.789,E2 -2844.789} C_VEL
LIN {X 0,Y 559.142,Z 314.454,A -85,B 0,C 180,E1 -2847.367,E2 -2847.367} C_VEL
LIN {X 0,Y 559.102,Z 314.465,A -85,B 0,C 180,E1 -2850.152,E2 -2850.152} C_VEL
LIN {X 0,Y 559.12,Z 314.458,A -85,B 0,C 180,E1 -2853.184,E2 -2853.184} C_VEL
LIN {X 0,Y 559.117,Z 314.459,A -85,B 0,C 180,E1 -2855.493,E2 -2855.493} C_VEL
LIN {X 0,Y 559.162,Z 314.454,A -85,B 0,C 180,E1 -2858.623,E2 -2858.623} C_VEL
LIN {X 0,Y 559.158,Z 314.453,A -85,B 0,C 180,E1 -2860.926,E2 -2860.926} C_VEL
LIN {X 0,Y 559.13,Z 314.461,A -85,B 0,C 180,E1 -2863.947,E2 -2863.947} C_VEL
LIN {X 0,Y 559.147,Z 314.463,A -85,B 0,C 180,E1 -2866.183,E2 -2866.183} C_VEL
LIN {X 0,Y 559.193,Z 314.443,A -85,B 0,C 180,E1 -2869.133,E2 -2869.133} C_VEL
LIN {X 0,Y 559.192,Z 314.455,A -85,B 0,C 180,E1 -2872.053,E2 -2872.053} C_VEL
LIN {X 0,Y 559.237,Z 314.443,A -85,B 0,C 180,E1 -2874.953,E2 -2874.953} C_VEL
LIN {X 0,Y 559.249,Z 314.447,A -85,B 0,C 180,E1 -2877.839,E2 -2877.839} C_VEL
LIN {X 0,Y 559.27,Z 314.439,A -85,B 0,C 180,E1 -2880.72,E2 -2880.72} C_VEL
LIN {X 0,Y 559.225,Z 314.445,A -85,B 0,C 180,E1 -2882.881,E2 -2882.881} C_VEL
LIN {X 0,Y 559.215,Z 314.451,A -85,B 0,C 180,E1 -2885.77,E2 -2885.77} C_VEL
LIN {X 0,Y 559.169,Z 314.453,A -85,B 0,C 180,E1 -2888.675,E2 -2888.675} C_VEL
LIN {X 0,Y 559.209,Z 314.451,A -85,B 0,C 180,E1 -2891.6,E2 -2891.6} C_VEL
LIN {X 0,Y 559.205,Z 314.448,A -85,B 0,C 180,E1 -2894.595,E2 -2894.595} C_VEL
LIN {X 0,Y 559.14,Z 314.46,A -85,B 0,C 180,E1 -2897.557,E2 -2897.557} C_VEL
LIN {X 0,Y 559.168,Z 314.462,A -85,B 0,C 180,E1 -2899.837,E2 -2899.837} C_VEL
LIN {X 0,Y 559.143,Z 314.46,A -85,B 0,C 180,E1 -2902.153,E2 -2902.153} C_VEL
LIN {X 0,Y 559.179,Z 314.454,A -85,B 0,C 180,E1 -2905.298,E2 -2905.298} C_VEL
LIN {X 0,Y 559.13,Z 314.467,A -85,B 0,C 180,E1 -2907.715,E2 -2907.715} C_VEL
LIN {X 0,Y 559.155,Z 314.457,A -85,B 0,C 180,E1 -2910.183,E2 -2910.183} C_VEL
LIN {X 0,Y 559.159,Z 314.453,A -85,B 0,C 180,E1 -2912.715,E2 -2912.715} C_VEL
LIN {X 0,Y 559.14,Z 314.461,A -85,B 0,C 180,E1 -2915.323,E2 -2915.323} C_VEL
LIN {X 0,Y 559.132,Z 314.46,A -85,B 0,C 180,E1 -2918.018,E2 -2918.018} C_VEL
LIN {X 0,Y 559.158,Z 314.454,A -85,B 0,C 180,E1 -2920.812,E2 -2920.812} C_VEL
LIN {X 0,Y 559.14,Z 314.463,A -85,B 0,C 180,E1 -2923.734,E2 -2923.734} C_VEL
LIN {X 0,Y 559.146,Z 314.456,A -85,B 0,C 180,E1 -2926.804,E2 -2926.804} C_VEL
LIN {X 0,Y 559.157,Z 314.459,A -85,B 0,C 180,E1 -2929.187,E2 -2929.187} C_VEL
LIN {X 0,Y 559.135,Z 314.46,A -85,B 0,C 180,E1 -2931.982,E2 -2931.982} C_VEL
LIN {X 0,Y 559.149,Z 314.457,A -85,B 0,C 180,E1 -2934.785,E2 -2934.785} C_VEL
LIN {X 0,Y 559.158,Z 314.464,A -85,B 0,C 180,E1 -2937.364,E2 -2937.364} C_VEL
LIN {X 0,Y 559.151,Z 314.456,A -85,B 0,C 180,E1 -2940.142,E2 -2940.142} C_VEL
LIN {X 0,Y 559.17,Z 314.46,A -85,B 0,C 180,E1 -2943.098,E2 -2943.098} C_VEL
LIN {X 0,Y 559.224,Z 314.51,A -85,B 0,C 180,E1 -2945.052,E2 -2945.052} C_VEL
LIN {X 0,Y 560.437,Z 320.608,A -85,B 0,C 180,E1 -2945.949,E2 -2945.949} C_VEL
LIN {X 0,Y 560.261,Z 334.908,A -85,B 0,C 180,E1 -2947.894,E2 -2947.894} C_VEL
LIN {X 0,Y 559.963,Z 355.212,A -85,B 0,C 180,E1 -2950.618,E2 -2950.618} C_VEL
LIN {X 0,Y 559.72,Z 371.62,A -85,B 0,C 180,E1 -2952.809,E2 -2952.809} C_VEL
LIN {X 0,Y 561.021,Z 379.079,A -85,B 0,C 180,E1 -2952.948,E2 -2952.948} C_VEL
LIN {X 0,Y 560.615,Z 508.627,A -85,B 0,C 180,E1 -2954.643,E2 -2954.643} C_VEL
LIN {X 0,Y 560.458,Z 523.102,A -85,B 0,C 180,E1 -2954.972,E2 -2954.972} C_VEL
LIN {X 0,Y 560.315,Z 536.501,A -85,B 0,C 180,E1 -2955.422,E2 -2955.422} C_VEL
LIN {X 0,Y 560.086,Z 549.874,A -85,B 0,C 180,E1 -2956.022,E2 -2956.022} C_VEL
LIN {X 0,Y 559.811,Z 562.675,A -85,B 0,C 180,E1 -2956.755,E2 -2956.755} C_VEL
LIN {X 0,Y 559.637,Z 574.31,A -85,B 0,C 180,E1 -2957.581,E2 -2957.581} C_VEL
LIN {X 0,Y 559.437,Z 584.883,A -85,B 0,C 180,E1 -2958.489,E2 -2958.489} C_VEL
LIN {X 0,Y 559.272,Z 594.706,A -85,B 0,C 180,E1 -2959.501,E2 -2959.501} C_VEL
LIN {X 0,Y 559.118,Z 603.557,A -85,B 0,C 180,E1 -2960.595,E2 -2960.595} C_VEL
LIN {X 0,Y 558.986,Z 612.035,A -85,B 0,C 180,E1 -2961.869,E2 -2961.869} C_VEL
LIN {X 0,Y 558.902,Z 618.865,A -85,B 0,C 180,E1 -2963.139,E2 -2963.139} C_VEL
LIN {X 0,Y 558.912,Z 623.569,A -85,B 0,C 180,E1 -2964.227,E2 -2964.227} C_VEL
LIN {X 0,Y 558.865,Z 628.444,A -85,B 0,C 180,E1 -2965.673,E2 -2965.673} C_VEL
LIN {X 0,Y 558.796,Z 631.832,A -85,B 0,C 180,E1 -2967.116,E2 -2967.116} C_VEL
LIN {X 0,Y 558.74,Z 633.833,A -85,B 0,C 180,E1 -2968.558,E2 -2968.558} C_VEL
LIN {X 0,Y 558.738,Z 634.5,A -85,B 0,C 180,E1 -2970,E2 -2970} C_VEL
LIN {X 0,Y 558.74,Z 633.834,A -85,B 0,C 180,E1 -2971.442,E2 -2971.442} C_VEL
LIN {X 0,Y 558.796,Z 631.834,A -85,B 0,C 180,E1 -2972.884,E2 -2972.884} C_VEL
LIN {X 0,Y 558.865,Z 628.446,A -85,B 0,C 180,E1 -2974.327,E2 -2974.327} C_VEL
LIN {X 0,Y 558.917,Z 623.568,A -85,B 0,C 180,E1 -2975.773,E2 -2975.773} C_VEL
LIN {X 0,Y 558.907,Z 617.053,A -85,B 0,C 180,E1 -2977.224,E2 -2977.224} C_VEL
LIN {X 0,Y 559.028,Z 609.801,A -85,B 0,C 180,E1 -2978.495,E2 -2978.495} C_VEL
LIN {X 0,Y 559.146,Z 600.821,A -85,B 0,C 180,E1 -2979.77,E2 -2979.77} C_VEL
LIN {X 0,Y 559.351,Z 591.391,A -85,B 0,C 180,E1 -2980.864,E2 -2980.864} C_VEL
LIN {X 0,Y 559.518,Z 580.952,A -85,B 0,C 180,E1 -2981.87,E2 -2981.87} C_VEL
LIN {X 0,Y 559.71,Z 569.43,A -85,B 0,C 180,E1 -2982.786,E2 -2982.786} C_VEL
LIN {X 0,Y 559.963,Z 556.639,A -85,B 0,C 180,E1 -2983.611,E2 -2983.611} C_VEL
LIN {X 0,Y 560.164,Z 544.146,A -85,B 0,C 180,E1 -2984.254,E2 -2984.254} C_VEL
LIN {X 0,Y 560.395,Z 531.071,A -85,B 0,C 180,E1 -2984.775,E2 -2984.775} C_VEL
LIN {X 0,Y 560.501,Z 517.582,A -85,B 0,C 180,E1 -2985.17,E2 -2985.17} C_VEL
LIN {X 0,Y 560.628,Z 502.591,A -85,B 0,C 180,E1 -2985.45,E2 -2985.45} C_VEL
LIN {X 0,Y 560.921,Z 378.215,A -85,B 0,C 180,E1 -2987.066,E2 -2987.066} C_VEL
LIN {X 0,Y 559.723,Z 371.6,A -85,B 0,C 180,E1 -2987.194,E2 -2987.194} C_VEL
LIN {X 0,Y 560.048,Z 350.619,A -85,B 0,C 180,E1 -2989.996,E2 -2989.996} C_VEL
LIN {X 0,Y 560.367,Z 330.589,A -85,B 0,C 180,E1 -2992.685,E2 -2992.685} C_VEL
LIN {X 0,Y 560.428,Z 320.594,A -85,B 0,C 180,E1 -2994.052,E2 -2994.052} C_VEL
LIN {X 0,Y 559.201,Z 314.459,A -85,B 0,C 180,E1 -2994.976,E2 -2994.976} C_VEL
LIN {X 0,Y 559.158,Z 314.456,A -85,B 0,C 180,E1 -2997.714,E2 -2997.714} C_VEL
LIN {X 0,Y 559.155,Z 314.457,A -85,B 0,C 180,E1 -3000.183,E2 -3000.183} C_VEL
LIN {X 0,Y 559.159,Z 314.462,A -85,B 0,C 180,E1 -3002.715,E2 -3002.715} C_VEL
LIN {X 0,Y 559.131,Z 314.458,A -85,B 0,C 180,E1 -3005.324,E2 -3005.324} C_VEL
LIN {X 0,Y 559.135,Z 314.459,A -85,B 0,C 180,E1 -3008.018,E2 -3008.018} C_VEL
LIN {X 0,Y 559.157,Z 314.458,A -85,B 0,C 180,E1 -3010.813,E2 -3010.813} C_VEL
LIN {X 0,Y 559.14,Z 314.456,A -85,B 0,C 180,E1 -3013.734,E2 -3013.734} C_VEL
LIN {X 0,Y 559.147,Z 314.459,A -85,B 0,C 180,E1 -3016.804,E2 -3016.804} C_VEL
LIN {X 0,Y 559.158,Z 314.454,A -85,B 0,C 180,E1 -3019.188,E2 -3019.188} C_VEL
LIN {X 0,Y 559.132,Z 314.46,A -85,B 0,C 180,E1 -3021.982,E2 -3021.982} C_VEL
LIN {X 0,Y 559.132,Z 314.46,A -85,B 0,C 180,E1 -3024.788,E2 -3024.788} C_VEL
LIN {X 0,Y 559.159,Z 314.453,A -85,B 0,C 180,E1 -3027.365,E2 -3027.365} C_VEL
LIN {X 0,Y 559.15,Z 314.462,A -85,B 0,C 180,E1 -3030.143,E2 -3030.143} C_VEL
LIN {X 0,Y 559.126,Z 314.457,A -85,B 0,C 180,E1 -3033.183,E2 -3033.183} C_VEL
LIN {X 0,Y 559.159,Z 314.454,A -85,B 0,C 180,E1 -3035.495,E2 -3035.495} C_VEL
LIN {X 0,Y 559.176,Z 314.454,A -85,B 0,C 180,E1 -3038.624,E2 -3038.624} C_VEL
LIN {X 0,Y 559.164,Z 314.453,A -85,B 0,C 180,E1 -3040.926,E2 -3040.926} C_VEL
LIN {X 0,Y 559.162,Z 314.46,A -85,B 0,C 180,E1 -3043.948,E2 -3043.948} C_VEL
LIN {X 0,Y 559.17,Z 314.458,A -85,B 0,C 180,E1 -3046.184,E2 -3046.184} C_VEL
LIN {X 0,Y 559.196,Z 314.449,A -85,B 0,C 180,E1 -3049.134,E2 -3049.134} C_VEL
LIN {X 0,Y 559.175,Z 314.459,A -85,B 0,C 180,E1 -3052.053,E2 -3052.053} C_VEL
LIN {X 0,Y 559.245,Z 314.442,A -85,B 0,C 180,E1 -3054.953,E2 -3054.953} C_VEL
LIN {X 0,Y 559.25,Z 314.449,A -85,B 0,C 180,E1 -3057.84,E2 -3057.84} C_VEL
LIN {X 0,Y 559.256,Z 314.448,A -85,B 0,C 180,E1 -3060,E2 -3060} C_VEL
LIN {X 0,Y 559.224,Z 314.444,A -85,B 0,C 180,E1 -3062.882,E2 -3062.882} C_VEL
LIN {X 0,Y 559.214,Z 314.456,A -85,B 0,C 180,E1 -3065.771,E2 -3065.771} C_VEL
LIN {X 0,Y 559.159,Z 314.453,A -85,B 0,C 180,E1 -3068.675,E2 -3068.675} C_VEL
LIN {X 0,Y 559.201,Z 314.455,A -85,B 0,C 180,E1 -3071.601,E2 -3071.601} C_VEL
LIN {X 0,Y 559.165,Z 314.453,A -85,B 0,C 180,E1 -3074.579,E2 -3074.579} C_VEL
LIN {X 0,Y 559.113,Z 314.466,A -85,B 0,C 180,E1 -3077.559,E2 -3077.559} C_VEL
LIN {X 0,Y 559.15,Z 314.46,A -85,B 0,C 180,E1 -3079.839,E2 -3079.839} C_VEL
LIN {X 0,Y 559.106,Z 314.462,A -85,B 0,C 180,E1 -3082.155,E2 -3082.155} C_VEL
LIN {X 0,Y 559.143,Z 314.458,A -85,B 0,C 180,E1 -3085.178,E2 -3085.178} C_VEL
LIN {X 0,Y 559.104,Z 314.466,A -85,B 0,C 180,E1 -3087.717,E2 -3087.717} C_VEL
LIN {X 0,Y 559.101,Z 314.456,A -85,B 0,C 180,E1 -3090.572,E2 -3090.572} C_VEL
LIN {X 0,Y 558.458,Z 314.542,A -85,B 0,C 180,E1 -3091.173,E2 -3091.173} C_VEL
LIN {X 0,Y 555.608,Z 314.896,A -85,B 0,C 180,E1 -3092.15,E2 -3092.15} C_VEL
LIN {X 0,Y 553.191,Z 315.198,A -85,B 0,C 180,E1 -3092.936,E2 -3092.936} C_VEL
LIN {X 0,Y 552.162,Z 315.333,A -85,B 0,C 180,E1 -3093.542,E2 -3093.542} C_VEL
LIN {X 0,Y 552.084,Z 315.335,A -85,B 0,C 180,E1 -3093.748,E2 -3093.748} C_VEL
LIN {X 0,Y 552.054,Z 315.335,A -85,B 0,C 180,E1 -3096.752,E2 -3096.752} C_VEL
LIN {X 0,Y 552.071,Z 315.343,A -85,B 0,C 180,E1 -3099.533,E2 -3099.533} C_VEL
LIN {X 0,Y 552.082,Z 315.335,A -85,B 0,C 180,E1 -3102.431,E2 -3102.431} C_VEL
LIN {X 0,Y 552.062,Z 315.343,A -85,B 0,C 180,E1 -3105.559,E2 -3105.559} C_VEL
LIN {X 0,Y 552.045,Z 315.341,A -85,B 0,C 180,E1 -3108.547,E2 -3108.547} C_VEL
LIN {X 0,Y 552.069,Z 315.345,A -85,B 0,C 180,E1 -3111.407,E2 -3111.407} C_VEL
LIN {X 0,Y 552.062,Z 315.34,A -85,B 0,C 180,E1 -3114.563,E2 -3114.563} C_VEL
LIN {X 0,Y 552.094,Z 315.343,A -85,B 0,C 180,E1 -3117.158,E2 -3117.158} C_VEL
LIN {X 0,Y 552.069,Z 315.339,A -85,B 0,C 180,E1 -3119.959,E2 -3119.959} C_VEL
LIN {X 0,Y 552.082,Z 315.345,A -85,B 0,C 180,E1 -3123.013,E2 -3123.013} C_VEL
LIN {X 0,Y 552.084,Z 315.348,A -85,B 0,C 180,E1 -3123.151,E2 -3123.151} C_VEL
LIN {X 0,Y 552.929,Z 320.216,A -85,B 0,C 180,E1 -3123.991,E2 -3123.991} C_VEL
LIN {X 0,Y 552.691,Z 337.454,A -85,B 0,C 180,E1 -3126.784,E2 -3126.784} C_VEL
LIN {X 0,Y 552.598,Z 342.735,A -85,B 0,C 180,E1 -3127.629,E2 -3127.629} C_VEL
LIN {X 0,Y 554.222,Z 351.887,A -85,B 0,C 180,E1 -3127.815,E2 -3127.815} C_VEL
LIN {X 0,Y 553.784,Z 479.033,A -85,B 0,C 180,E1 -3129.501,E2 -3129.501} C_VEL
LIN {X 0,Y 553.614,Z 493.315,A -85,B 0,C 180,E1 -3129.834,E2 -3129.834} C_VEL
LIN {X 0,Y 553.441,Z 506.853,A -85,B 0,C 180,E1 -3130.297,E2 -3130.297} C_VEL
LIN {X 0,Y 553.18,Z 520.16,A -85,B 0,C 180,E1 -3130.904,E2 -3130.904} C_VEL
LIN {X 0,Y 552.914,Z 533.161,A -85,B 0,C 180,E1 -3131.664,E2 -3131.664} C_VEL
LIN {X 0,Y 552.666,Z 544.798,A -85,B 0,C 180,E1 -3132.506,E2 -3132.506} C_VEL
LIN {X 0,Y 552.449,Z 554.683,A -85,B 0,C 180,E1 -3133.367,E2 -3133.367} C_VEL
LIN {X 0,Y 552.229,Z 565.476,A -85,B 0,C 180,E1 -3134.499,E2 -3134.499} C_VEL
LIN {X 0,Y 552.029,Z 574.729,A -85,B 0,C 180,E1 -3135.678,E2 -3135.678} C_VEL
LIN {X 0,Y 551.887,Z 582.801,A -85,B 0,C 180,E1 -3136.936,E2 -3136.936} C_VEL
LIN {X 0,Y 551.805,Z 589.555,A -85,B 0,C 180,E1 -3138.242,E2 -3138.242} C_VEL
LIN {X 0,Y 551.735,Z 595.517,A -85,B 0,C 180,E1 -3139.727,E2 -3139.727} C_VEL
LIN {X 0,Y 551.695,Z 599.866,A -85,B 0,C 180,E1 -3141.207,E2 -3141.207} C_VEL
LIN {X 0,Y 551.694,Z 602.741,A -85,B 0,C 180,E1 -3142.681,E2 -3142.681} C_VEL
LIN {X 0,Y 551.706,Z 604.23,A -85,B 0,C 180,E1 -3144.151,E2 -3144.151} C_VEL
LIN {X 0,Y 551.694,Z 604.382,A -85,B 0,C 180,E1 -3145.616,E2 -3145.616} C_VEL
LIN {X 0,Y 551.712,Z 603.208,A -85,B 0,C 180,E1 -3147.079,E2 -3147.079} C_VEL
LIN {X 0,Y 551.65,Z 600.69,A -85,B 0,C 180,E1 -3148.54,E2 -3148.54} C_VEL
LIN {X 0,Y 551.686,Z 596.745,A -85,B 0,C 180,E1 -3150,E2 -3150} C_VEL
LIN {X 0,Y 551.825,Z 592.786,A -85,B 0,C 180,E1 -3151.095,E2 -3151.095} C_VEL
LIN {X 0,Y 551.772,Z 587.905,A -85,B 0,C 180,E1 -3152.19,E2 -3152.19} C_VEL
LIN {X 0,Y 551.951,Z 580.905,A -85,B 0,C 180,E1 -3153.467,E2 -3153.467} C_VEL
LIN {X 0,Y 552.13,Z 572.268,A -85,B 0,C 180,E1 -3154.746,E2 -3154.746} C_VEL
LIN {X 0,Y 552.305,Z 563.258,A -85,B 0,C 180,E1 -3155.843,E2 -3155.843} C_VEL
LIN {X 0,Y 552.513,Z 552.961,A -85,B 0,C 180,E1 -3156.886,E2 -3156.886} C_VEL
LIN {X 0,Y 552.753,Z 541.335,A -85,B 0,C 180,E1 -3157.856,E2 -3157.856} C_VEL
LIN {X 0,Y 552.989,Z 529.177,A -85,B 0,C 180,E1 -3158.68,E2 -3158.68} C_VEL
LIN {X 0,Y 553.227,Z 517.536,A -85,B 0,C 180,E1 -3159.321,E2 -3159.321} C_VEL
LIN {X 0,Y 553.446,Z 503.643,A -85,B 0,C 180,E1 -3159.917,E2 -3159.917} C_VEL
LIN {X 0,Y 553.641,Z 489.744,A -85,B 0,C 180,E1 -3160.352,E2 -3160.352} C_VEL
LIN {X 0,Y 553.79,Z 475.17,A -85,B 0,C 180,E1 -3160.65,E2 -3160.65} C_VEL
LIN {X 0,Y 554.11,Z 350.669,A -85,B 0,C 180,E1 -3162.295,E2 -3162.295} C_VEL
LIN {X 0,Y 552.598,Z 342.749,A -85,B 0,C 180,E1 -3162.46,E2 -3162.46} C_VEL
LIN {X 0,Y 552.927,Z 325.107,A -85,B 0,C 180,E1 -3165.306,E2 -3165.306} C_VEL
LIN {X 0,Y 552.865,Z 319.393,A -85,B 0,C 180,E1 -3166.24,E2 -3166.24} C_VEL
LIN {X 0,Y 552.136,Z 315.338,A -85,B 0,C 180,E1 -3166.976,E2 -3166.976} C_VEL
LIN {X 0,Y 552.094,Z 315.336,A -85,B 0,C 180,E1 -3170.103,E2 -3170.103} C_VEL
LIN {X 0,Y 552.052,Z 315.343,A -85,B 0,C 180,E1 -3172.453,E2 -3172.453} C_VEL
LIN {X 0,Y 552.062,Z 315.342,A -85,B 0,C 180,E1 -3175.328,E2 -3175.328} C_VEL
LIN {X 0,Y 552.048,Z 315.341,A -85,B 0,C 180,E1 -3178.102,E2 -3178.102} C_VEL
LIN {X 0,Y 552.064,Z 315.343,A -85,B 0,C 180,E1 -3180.612,E2 -3180.612} C_VEL
LIN {X 0,Y 552.052,Z 315.343,A -85,B 0,C 180,E1 -3183.19,E2 -3183.19} C_VEL
LIN {X 0,Y 552.067,Z 315.337,A -85,B 0,C 180,E1 -3185.845,E2 -3185.845} C_VEL
LIN {X 0,Y 552.072,Z 315.341,A -85,B 0,C 180,E1 -3189.054,E2 -3189.054} C_VEL
LIN {X 0,Y 552.054,Z 315.339,A -85,B 0,C 180,E1 -3191.452,E2 -3191.452} C_VEL
LIN {X 0,Y 552.064,Z 315.345,A -85,B 0,C 180,E1 -3194.528,E2 -3194.528} C_VEL
LIN {X 0,Y 552.082,Z 315.335,A -85,B 0,C 180,E1 -3197.591,E2 -3197.591} C_VEL
LIN {X 0,Y 552.073,Z 315.34,A -85,B 0,C 180,E1 -3200.946,E2 -3200.946} C_VEL
LIN {X 0,Y 552.054,Z 315.338,A -85,B 0,C 180,E1 -3203.325,E2 -3203.325} C_VEL
LIN {X 0,Y 552.099,Z 315.335,A -85,B 0,C 180,E1 -3205.937,E2 -3205.937} C_VEL
LIN {X 0,Y 552.091,Z 315.343,A -85,B 0,C 180,E1 -3208.538,E2 -3208.538} C_VEL
LIN {X 0,Y 552.075,Z 315.335,A -85,B 0,C 180,E1 -3211.448,E2 -3211.448} C_VEL
LIN {X 0,Y 552.085,Z 315.342,A -85,B 0,C 180,E1 -3214.353,E2 -3214.353} C_VEL
LIN {X 0,Y 552.049,Z 315.342,A -85,B 0,C 180,E1 -3216.755,E2 -3216.755} C_VEL
LIN {X 0,Y 552.099,Z 315.328,A -85,B 0,C 180,E1 -3219.119,E2 -3219.119} C_VEL
LIN {X 0,Y 552.082,Z 315.332,A -85,B 0,C 180,E1 -3221.443,E2 -3221.443} C_VEL
LIN {X 0,Y 552.09,Z 315.34,A -85,B 0,C 180,E1 -3224.495,E2 -3224.495} C_VEL
LIN {X 0,Y 552.102,Z 315.332,A -85,B 0,C 180,E1 -3226.754,E2 -3226.754} C_VEL
LIN {X 0,Y 552.163,Z 315.319,A -85,B 0,C 180,E1 -3228.993,E2 -3228.993} C_VEL
LIN {X 0,Y 552.147,Z 315.33,A -85,B 0,C 180,E1 -3231.951,E2 -3231.951} C_VEL
LIN {X 0,Y 552.214,Z 315.319,A -85,B 0,C 180,E1 -3234.889,E2 -3234.889} C_VEL
LIN {X 0,Y 552.221,Z 315.322,A -85,B 0,C 180,E1 -3237.812,E2 -3237.812} C_VEL
LIN {X 0,Y 552.24,Z 315.315,A -85,B 0,C 180,E1 -3240.729,E2 -3240.729} C_VEL
LIN {X 0,Y 552.191,Z 315.321,A -85,B 0,C 180,E1 -3242.918,E2 -3242.918} C_VEL
LIN {X 0,Y 552.186,Z 315.328,A -85,B 0,C 180,E1 -3245.844,E2 -3245.844} C_VEL
LIN {X 0,Y 552.14,Z 315.328,A -85,B 0,C 180,E1 -3248.786,E2 -3248.786} C_VEL
LIN {X 0,Y 552.165,Z 315.331,A -85,B 0,C 180,E1 -3251.75,E2 -3251.75} C_VEL
LIN {X 0,Y 552.14,Z 315.327,A -85,B 0,C 180,E1 -3254.748,E2 -3254.748} C_VEL
LIN {X 0,Y 552.098,Z 315.341,A -85,B 0,C 180,E1 -3257.789,E2 -3257.789} C_VEL
LIN {X 0,Y 552.129,Z 315.335,A -85,B 0,C 180,E1 -3260.101,E2 -3260.101} C_VEL
LIN {X 0,Y 552.094,Z 315.334,A -85,B 0,C 180,E1 -3262.451,E2 -3262.451} C_VEL
LIN {X 0,Y 552.141,Z 315.331,A -85,B 0,C 180,E1 -3265.346,E2 -3265.346} C_VEL
LIN {X 0,Y 552.081,Z 315.339,A -85,B 0,C 180,E1 -3268.1,E2 -3268.1} C_VEL
LIN {X 0,Y 552.104,Z 315.333,A -85,B 0,C 180,E1 -3270.609,E2 -3270.609} C_VEL
LIN {X 0,Y 552.118,Z 315.333,A -85,B 0,C 180,E1 -3273.186,E2 -3273.186} C_VEL
LIN {X 0,Y 552.09,Z 315.341,A -85,B 0,C 180,E1 -3275.843,E2 -3275.843} C_VEL
LIN {X 0,Y 552.122,Z 315.332,A -85,B 0,C 180,E1 -3279.061,E2 -3279.061} C_VEL
LIN {X 0,Y 552.123,Z 315.338,A -85,B 0,C 180,E1 -3281.446,E2 -3281.446} C_VEL
LIN {X 0,Y 552.091,Z 315.334,A -85,B 0,C 180,E1 -3284.531,E2 -3284.531} C_VEL
LIN {X 0,Y 552.132,Z 315.337,A -85,B 0,C 180,E1 -3287.584,E2 -3287.584} C_VEL
LIN {X 0,Y 552.131,Z 315.33,A -85,B 0,C 180,E1 -3290.473,E2 -3290.473} C_VEL
LIN {X 0,Y 552.114,Z 315.34,A -85,B 0,C 180,E1 -3293.316,E2 -3293.316} C_VEL
LIN {X 0,Y 552.131,Z 315.333,A -85,B 0,C 180,E1 -3295.939,E2 -3295.939} C_VEL
LIN {X 0,Y 552.121,Z 315.331,A -85,B 0,C 180,E1 -3298.541,E2 -3298.541} C_VEL
LIN {X 0,Y 552.127,Z 315.338,A -85,B 0,C 180,E1 -3301.438,E2 -3301.438} C_VEL
LIN {X 0,Y 552.132,Z 315.333,A -85,B 0,C 180,E1 -3304.356,E2 -3304.356} C_VEL
LIN {X 0,Y 552.163,Z 315.379,A -85,B 0,C 180,E1 -3304.857,E2 -3304.857} C_VEL
LIN {X 0,Y 553.519,Z 321.865,A -85,B 0,C 180,E1 -3305.828,E2 -3305.828} C_VEL
LIN {X 0,Y 553.36,Z 335.766,A -85,B 0,C 180,E1 -3307.745,E2 -3307.745} C_VEL
LIN {X 0,Y 553.007,Z 356.46,A -85,B 0,C 180,E1 -3310.553,E2 -3310.553} C_VEL
LIN {X 0,Y 552.789,Z 371.552,A -85,B 0,C 180,E1 -3312.577,E2 -3312.577} C_VEL
LIN {X 0,Y 554.227,Z 380.015,A -85,B 0,C 180,E1 -3312.745,E2 -3312.745} C_VEL
LIN {X 0,Y 553.778,Z 508.627,A -85,B 0,C 180,E1 -3314.449,E2 -3314.449} C_VEL
LIN {X 0,Y 553.573,Z 523.285,A -85,B 0,C 180,E1 -3314.786,E2 -3314.786} C_VEL
LIN {X 0,Y 553.43,Z 536.612,A -85,B 0,C 180,E1 -3315.241,E2 -3315.241} C_VEL
LIN {X 0,Y 553.185,Z 549.872,A -85,B 0,C 180,E1 -3315.844,E2 -3315.844} C_VEL
LIN {X 0,Y 552.888,Z 562.673,A -85,B 0,C 180,E1 -3316.586,E2 -3316.586} C_VEL
LIN {X 0,Y 552.646,Z 574.308,A -85,B 0,C 180,E1 -3317.421,E2 -3317.421} C_VEL
LIN {X 0,Y 552.446,Z 585.468,A -85,B 0,C 180,E1 -3318.397,E2 -3318.397} C_VEL
LIN {X 0,Y 552.252,Z 594.706,A -85,B 0,C 180,E1 -3319.366,E2 -3319.366} C_VEL
LIN {X 0,Y 552.069,Z 603.557,A -85,B 0,C 180,E1 -3320.474,E2 -3320.474} C_VEL
LIN {X 0,Y 551.927,Z 612.035,A -85,B 0,C 180,E1 -3321.764,E2 -3321.764} C_VEL
LIN {X 0,Y 551.823,Z 618.863,A -85,B 0,C 180,E1 -3323.051,E2 -3323.051} C_VEL
LIN {X 0,Y 551.792,Z 624.961,A -85,B 0,C 180,E1 -3324.518,E2 -3324.518} C_VEL
LIN {X 0,Y 551.759,Z 628.444,A -85,B 0,C 180,E1 -3325.617,E2 -3325.617} C_VEL
LIN {X 0,Y 551.72,Z 631.832,A -85,B 0,C 180,E1 -3327.079,E2 -3327.079} C_VEL
LIN {X 0,Y 551.64,Z 633.834,A -85,B 0,C 180,E1 -3328.54,E2 -3328.54} C_VEL
LIN {X 0,Y 551.639,Z 634.5,A -85,B 0,C 180,E1 -3330,E2 -3330} C_VEL
LIN {X 0,Y 551.64,Z 633.835,A -85,B 0,C 180,E1 -3331.46,E2 -3331.46} C_VEL
LIN {X 0,Y 551.72,Z 631.835,A -85,B 0,C 180,E1 -3332.921,E2 -3332.921} C_VEL
LIN {X 0,Y 551.759,Z 628.446,A -85,B 0,C 180,E1 -3334.383,E2 -3334.383} C_VEL
LIN {X 0,Y 551.825,Z 623.567,A -85,B 0,C 180,E1 -3335.848,E2 -3335.848} C_VEL
LIN {X 0,Y 551.833,Z 617.054,A -85,B 0,C 180,E1 -3337.317,E2 -3337.317} C_VEL
LIN {X 0,Y 551.963,Z 609.802,A -85,B 0,C 180,E1 -3338.604,E2 -3338.604} C_VEL
LIN {X 0,Y 552.116,Z 600.821,A -85,B 0,C 180,E1 -3339.895,E2 -3339.895} C_VEL
LIN {X 0,Y 552.346,Z 591.391,A -85,B 0,C 180,E1 -3341.003,E2 -3341.003} C_VEL
LIN {X 0,Y 552.539,Z 580.952,A -85,B 0,C 180,E1 -3342.022,E2 -3342.022} C_VEL
LIN {X 0,Y 552.761,Z 569.428,A -85,B 0,C 180,E1 -3342.95,E2 -3342.95} C_VEL
LIN {X 0,Y 553.026,Z 556.637,A -85,B 0,C 180,E1 -3343.785,E2 -3343.785} C_VEL
LIN {X 0,Y 553.286,Z 544.143,A -85,B 0,C 180,E1 -3344.435,E2 -3344.435} C_VEL
LIN {X 0,Y 553.53,Z 531.063,A -85,B 0,C 180,E1 -3344.963,E2 -3344.963} C_VEL
LIN {X 0,Y 553.668,Z 517.439,A -85,B 0,C 180,E1 -3345.366,E2 -3345.366} C_VEL
LIN {X 0,Y 553.799,Z 502.591,A -85,B 0,C 180,E1 -3345.645,E2 -3345.645} C_VEL
LIN {X 0,Y 554.164,Z 379.101,A -85,B 0,C 180,E1 -3347.269,E2 -3347.269} C_VEL
LIN {X 0,Y 552.779,Z 371.516,A -85,B 0,C 180,E1 -3347.428,E2 -3347.428} C_VEL
LIN {X 0,Y 553.104,Z 351.852,A -85,B 0,C 180,E1 -3350.064,E2 -3350.064} C_VEL
LIN {X 0,Y 553.459,Z 331.827,A -85,B 0,C 180,E1 -3352.787,E2 -3352.787} C_VEL
LIN {X 0,Y 553.511,Z 321.855,A -85,B 0,C 180,E1 -3354.173,E2 -3354.173} C_VEL
LIN {X 0,Y 552.16,Z 315.334,A -85,B 0,C 180,E1 -3355.175,E2 -3355.175} C_VEL
LIN {X 0,Y 552.111,Z 315.336,A -85,B 0,C 180,E1 -3358.098,E2 -3358.098} C_VEL
LIN {X 0,Y 552.104,Z 315.339,A -85,B 0,C 180,E1 -3360.609,E2 -3360.609} C_VEL
LIN {X 0,Y 552.118,Z 315.332,A -85,B 0,C 180,E1 -3363.186,E2 -3363.186} C_VEL
LIN {X 0,Y 552.089,Z 315.336,A -85,B 0,C 180,E1 -3365.844,E2 -3365.844} C_VEL
LIN {X 0,Y 552.123,Z 315.332,A -85,B 0,C 180,E1 -3369.061,E2 -3369.061} C_VEL
LIN {X 0,Y 552.122,Z 315.33,A -85,B 0,C 180,E1 -3371.446,E2 -3371.446} C_VEL
LIN {X 0,Y 552.091,Z 315.342,A -85,B 0,C 180,E1 -3374.531,E2 -3374.531} C_VEL
LIN {X 0,Y 552.132,Z 315.329,A -85,B 0,C 180,E1 -3377.585,E2 -3377.585} C_VEL
LIN {X 0,Y 552.131,Z 315.337,A -85,B 0,C 180,E1 -3380.473,E2 -3380.473} C_VEL
LIN {X 0,Y 552.101,Z 315.332,A -85,B 0,C 180,E1 -3383.318,E2 -3383.318} C_VEL
LIN {X 0,Y 552.129,Z 315.333,A -85,B 0,C 180,E1 -3385.939,E2 -3385.939} C_VEL
LIN {X 0,Y 552.123,Z 315.335,A -85,B 0,C 180,E1 -3388.541,E2 -3388.541} C_VEL
LIN {X 0,Y 552.101,Z 315.333,A -85,B 0,C 180,E1 -3391.444,E2 -3391.444} C_VEL
LIN {X 0,Y 552.14,Z 315.331,A -85,B 0,C 180,E1 -3394.654,E2 -3394.654} C_VEL
LIN {X 0,Y 552.094,Z 315.334,A -85,B 0,C 180,E1 -3397.549,E2 -3397.549} C_VEL
LIN {X 0,Y 552.149,Z 315.332,A -85,B 0,C 180,E1 -3400.375,E2 -3400.375} C_VEL
LIN {X 0,Y 552.136,Z 315.328,A -85,B 0,C 180,E1 -3402.977,E2 -3402.977} C_VEL
LIN {X 0,Y 552.136,Z 315.337,A -85,B 0,C 180,E1 -3406.005,E2 -3406.005} C_VEL
LIN {X 0,Y 552.165,Z 315.325,A -85,B 0,C 180,E1 -3408.994,E2 -3408.994} C_VEL
LIN {X 0,Y 552.136,Z 315.335,A -85,B 0,C 180,E1 -3411.951,E2 -3411.951} C_VEL
LIN {X 0,Y 552.22,Z 315.318,A -85,B 0,C 180,E1 -3414.889,E2 -3414.889} C_VEL
LIN {X 0,Y 552.222,Z 315.323,A -85,B 0,C 180,E1 -3417.812,E2 -3417.812} C_VEL
LIN {X 0,Y 552.225,Z 315.324,A -85,B 0,C 180,E1 -3420,E2 -3420} C_VEL
LIN {X 0,Y 552.193,Z 315.32,A -85,B 0,C 180,E1 -3422.918,E2 -3422.918} C_VEL
LIN {X 0,Y 552.182,Z 315.33,A -85,B 0,C 180,E1 -3425.844,E2 -3425.844} C_VEL
LIN {X 0,Y 552.133,Z 315.329,A -85,B 0,C 180,E1 -3428.786,E2 -3428.786} C_VEL
LIN {X 0,Y 552.155,Z 315.333,A -85,B 0,C 180,E1 -3431.751,E2 -3431.751} C_VEL
LIN {X 0,Y 552.126,Z 315.329,A -85,B 0,C 180,E1 -3434.749,E2 -3434.749} C_VEL
LIN {X 0,Y 552.079,Z 315.343,A -85,B 0,C 180,E1 -3437.79,E2 -3437.79} C_VEL
LIN {X 0,Y 552.101,Z 315.334,A -85,B 0,C 180,E1 -3440.103,E2 -3440.103} C_VEL
LIN {X 0,Y 552.046,Z 315.34,A -85,B 0,C 180,E1 -3442.453,E2 -3442.453} C_VEL
LIN {X 0,Y 552.087,Z 315.339,A -85,B 0,C 180,E1 -3445.334,E2 -3445.334} C_VEL
LIN {X 0,Y 552.052,Z 315.339,A -85,B 0,C 180,E1 -3448.102,E2 -3448.102} C_VEL
LIN {X 0,Y 552.071,Z 315.331,A -85,B 0,C 180,E1 -3450.612,E2 -3450.612} C_VEL
LIN {X 0,Y 552.099,Z 315.337,A -85,B 0,C 180,E1 -3453.187,E2 -3453.187} C_VEL
LIN {X 0,Y 552.084,Z 315.335,A -85,B 0,C 180,E1 -3453.748,E2 -3453.748} C_VEL
LIN {X 0,Y 551.428,Z 315.419,A -85,B 0,C 180,E1 -3454.357,E2 -3454.357} C_VEL
LIN {X 0,Y 548.562,Z 315.781,A -85,B 0,C 180,E1 -3455.345,E2 -3455.345} C_VEL
LIN {X 0,Y 546.13,Z 316.076,A -85,B 0,C 180,E1 -3456.14,E2 -3456.14} C_VEL
LIN {X 0,Y 545.085,Z 316.203,A -85,B 0,C 180,E1 -3456.754,E2 -3456.754} C_VEL
LIN {X 0,Y 545.001,Z 316.215,A -85,B 0,C 180,E1 -3456.962,E2 -3456.962} C_VEL
LIN {X 0,Y 545.023,Z 316.223,A -85,B 0,C 180,E1 -3459.313,E2 -3459.313} C_VEL
LIN {X 0,Y 545.032,Z 316.214,A -85,B 0,C 180,E1 -3462.108,E2 -3462.108} C_VEL
LIN {X 0,Y 545.013,Z 316.224,A -85,B 0,C 180,E1 -3465.173,E2 -3465.173} C_VEL
LIN {X 0,Y 545.028,Z 316.216,A -85,B 0,C 180,E1 -3467.892,E2 -3467.892} C_VEL
LIN {X 0,Y 545.03,Z 316.218,A -85,B 0,C 180,E1 -3470.814,E2 -3470.814} C_VEL
LIN {X 0,Y 545.003,Z 316.221,A -85,B 0,C 180,E1 -3473.616,E2 -3473.616} C_VEL
LIN {X 0,Y 545.031,Z 316.214,A -85,B 0,C 180,E1 -3476.325,E2 -3476.325} C_VEL
LIN {X 0,Y 545.035,Z 316.22,A -85,B 0,C 180,E1 -3478.95,E2 -3478.95} C_VEL
LIN {X 0,Y 545.036,Z 316.22,A -85,B 0,C 180,E1 -3481.504,E2 -3481.504} C_VEL
LIN {X 0,Y 545.068,Z 316.315,A -85,B 0,C 180,E1 -3482.985,E2 -3482.985} C_VEL
LIN {X 0,Y 546.023,Z 322.419,A -85,B 0,C 180,E1 -3484.047,E2 -3484.047} C_VEL
LIN {X 0,Y 545.692,Z 339.66,A -85,B 0,C 180,E1 -3486.87,E2 -3486.87} C_VEL
LIN {X 0,Y 545.649,Z 342.977,A -85,B 0,C 180,E1 -3487.408,E2 -3487.408} C_VEL
LIN {X 0,Y 547.47,Z 353.125,A -85,B 0,C 180,E1 -3487.609,E2 -3487.609} C_VEL
LIN {X 0,Y 546.964,Z 479.398,A -85,B 0,C 180,E1 -3489.307,E2 -3489.307} C_VEL
LIN {X 0,Y 546.752,Z 493.542,A -85,B 0,C 180,E1 -3489.643,E2 -3489.643} C_VEL
LIN {X 0,Y 546.544,Z 506.56,A -85,B 0,C 180,E1 -3490.093,E2 -3490.093} C_VEL
LIN {X 0,Y 546.32,Z 518.911,A -85,B 0,C 180,E1 -3490.655,E2 -3490.655} C_VEL
LIN {X 0,Y 546.012,Z 532.139,A -85,B 0,C 180,E1 -3491.423,E2 -3491.423} C_VEL
LIN {X 0,Y 545.736,Z 543.639,A -85,B 0,C 180,E1 -3492.251,E2 -3492.251} C_VEL
LIN {X 0,Y 545.471,Z 553.983,A -85,B 0,C 180,E1 -3493.148,E2 -3493.148} C_VEL
LIN {X 0,Y 545.208,Z 564.893,A -85,B 0,C 180,E1 -3494.294,E2 -3494.294} C_VEL
LIN {X 0,Y 545.009,Z 574.568,A -85,B 0,C 180,E1 -3495.535,E2 -3495.535} C_VEL
LIN {X 0,Y 544.823,Z 582.41,A -85,B 0,C 180,E1 -3496.764,E2 -3496.764} C_VEL
LIN {X 0,Y 544.733,Z 589.257,A -85,B 0,C 180,E1 -3498.087,E2 -3498.087} C_VEL
LIN {X 0,Y 544.692,Z 593.938,A -85,B 0,C 180,E1 -3499.217,E2 -3499.217} C_VEL
LIN {X 0,Y 544.62,Z 598.77,A -85,B 0,C 180,E1 -3500.717,E2 -3500.717} C_VEL
LIN {X 0,Y 544.62,Z 601.353,A -85,B 0,C 180,E1 -3501.839,E2 -3501.839} C_VEL
LIN {X 0,Y 544.652,Z 603.584,A -85,B 0,C 180,E1 -3503.331,E2 -3503.331} C_VEL
LIN {X 0,Y 544.596,Z 604.458,A -85,B 0,C 180,E1 -3504.817,E2 -3504.817} C_VEL
LIN {X 0,Y 544.627,Z 604.002,A -85,B 0,C 180,E1 -3506.301,E2 -3506.301} C_VEL
LIN {X 0,Y 544.57,Z 602.219,A -85,B 0,C 180,E1 -3507.781,E2 -3507.781} C_VEL
LIN {X 0,Y 544.553,Z 599.074,A -85,B 0,C 180,E1 -3509.26,E2 -3509.26} C_VEL
LIN {X 0,Y 544.608,Z 594.454,A -85,B 0,C 180,E1 -3510.739,E2 -3510.739} C_VEL
LIN {X 0,Y 544.685,Z 588.22,A -85,B 0,C 180,E1 -3512.218,E2 -3512.218} C_VEL
LIN {X 0,Y 544.875,Z 581.293,A -85,B 0,C 180,E1 -3513.513,E2 -3513.513} C_VEL
LIN {X 0,Y 545.086,Z 572.737,A -85,B 0,C 180,E1 -3514.807,E2 -3514.807} C_VEL
LIN {X 0,Y 545.274,Z 563.823,A -85,B 0,C 180,E1 -3515.918,E2 -3515.918} C_VEL
LIN {X 0,Y 545.515,Z 553.829,A -85,B 0,C 180,E1 -3516.956,E2 -3516.956} C_VEL
LIN {X 0,Y 545.765,Z 542.168,A -85,B 0,C 180,E1 -3517.957,E2 -3517.957} C_VEL
LIN {X 0,Y 546.048,Z 530.241,A -85,B 0,C 180,E1 -3518.792,E2 -3518.792} C_VEL
LIN {X 0,Y 546.298,Z 518.821,A -85,B 0,C 180,E1 -3519.441,E2 -3519.441} C_VEL
LIN {X 0,Y 546.574,Z 505.451,A -85,B 0,C 180,E1 -3520.043,E2 -3520.043} C_VEL
LIN {X 0,Y 546.813,Z 491.415,A -85,B 0,C 180,E1 -3520.507,E2 -3520.507} C_VEL
LIN {X 0,Y 546.957,Z 477.894,A -85,B 0,C 180,E1 -3520.808,E2 -3520.808} C_VEL
LIN {X 0,Y 547.353,Z 351.765,A -85,B 0,C 180,E1 -3522.503,E2 -3522.503} C_VEL
LIN {X 0,Y 545.652,Z 342.892,A -85,B 0,C 180,E1 -3522.695,E2 -3522.695} C_VEL
LIN {X 0,Y 546.056,Z 324.598,A -85,B 0,C 180,E1 -3525.681,E2 -3525.681} C_VEL
LIN {X 0,Y 545.805,Z 319.979,A -85,B 0,C 180,E1 -3526.456,E2 -3526.456} C_VEL
LIN {X 0,Y 545.072,Z 316.218,A -85,B 0,C 180,E1 -3527.154,E2 -3527.154} C_VEL
LIN {X 0,Y 545.033,Z 316.218,A -85,B 0,C 180,E1 -3530.375,E2 -3530.375} C_VEL
LIN {X 0,Y 545.01,Z 316.224,A -85,B 0,C 180,E1 -3532.759,E2 -3532.759} C_VEL
LIN {X 0,Y 545.007,Z 316.22,A -85,B 0,C 180,E1 -3535.488,E2 -3535.488} C_VEL
LIN {X 0,Y 544.997,Z 316.219,A -85,B 0,C 180,E1 -3537.661,E2 -3537.661} C_VEL
LIN {X 0,Y 545.023,Z 316.216,A -85,B 0,C 180,E1 -3540.235,E2 -3540.235} C_VEL
LIN {X 0,Y 545.04,Z 316.218,A -85,B 0,C 180,E1 -3543.055,E2 -3543.055} C_VEL
LIN {X 0,Y 545.017,Z 316.215,A -85,B 0,C 180,E1 -3545.67,E2 -3545.67} C_VEL
LIN {X 0,Y 545.017,Z 316.218,A -85,B 0,C 180,E1 -3548.241,E2 -3548.241} C_VEL
LIN {X 0,Y 545.004,Z 316.22,A -85,B 0,C 180,E1 -3551.122,E2 -3551.122} C_VEL
LIN {X 0,Y 545.024,Z 316.217,A -85,B 0,C 180,E1 -3554.133,E2 -3554.133} C_VEL
LIN {X 0,Y 545.001,Z 316.222,A -85,B 0,C 180,E1 -3556.885,E2 -3556.885} C_VEL
LIN {X 0,Y 545,Z 316.217,A -85,B 0,C 180,E1 -3559.538,E2 -3559.538} C_VEL
LIN {X 0,Y 545.022,Z 316.215,A -85,B 0,C 180,E1 -3561.868,E2 -3561.868} C_VEL
LIN {X 0,Y 545.025,Z 316.223,A -85,B 0,C 180,E1 -3564.53,E2 -3564.53} C_VEL
LIN {X 0,Y 545.056,Z 316.209,A -85,B 0,C 180,E1 -3567.21,E2 -3567.21} C_VEL
LIN {X 0,Y 545.023,Z 316.215,A -85,B 0,C 180,E1 -3569.808,E2 -3569.808} C_VEL
LIN {X 0,Y 545.027,Z 316.216,A -85,B 0,C 180,E1 -3572.841,E2 -3572.841} C_VEL
LIN {X 0,Y 545.021,Z 316.215,A -85,B 0,C 180,E1 -3575.629,E2 -3575.629} C_VEL
LIN {X 0,Y 545.038,Z 316.209,A -85,B 0,C 180,E1 -3578.835,E2 -3578.835} C_VEL
LIN {X 0,Y 545.046,Z 316.209,A -85,B 0,C 180,E1 -3581.194,E2 -3581.194} C_VEL
LIN {X 0,Y 545.037,Z 316.222,A -85,B 0,C 180,E1 -3584.289,E2 -3584.289} C_VEL
LIN {X 0,Y 545.052,Z 316.212,A -85,B 0,C 180,E1 -3586.579,E2 -3586.579} C_VEL
LIN {X 0,Y 545.119,Z 316.197,A -85,B 0,C 180,E1 -3588.849,E2 -3588.849} C_VEL
LIN {X 0,Y 545.096,Z 316.207,A -85,B 0,C 180,E1 -3591.846,E2 -3591.846} C_VEL
LIN {X 0,Y 545.172,Z 316.196,A -85,B 0,C 180,E1 -3594.822,E2 -3594.822} C_VEL
LIN {X 0,Y 545.193,Z 316.197,A -85,B 0,C 180,E1 -3597.783,E2 -3597.783} C_VEL
LIN {X 0,Y 545.211,Z 316.19,A -85,B 0,C 180,E1 -3600.738,E2 -3600.738} C_VEL
LIN {X 0,Y 545.157,Z 316.198,A -85,B 0,C 180,E1 -3602.956,E2 -3602.956} C_VEL
LIN {X 0,Y 545.136,Z 316.207,A -85,B 0,C 180,E1 -3605.92,E2 -3605.92} C_VEL
LIN {X 0,Y 545.101,Z 316.204,A -85,B 0,C 180,E1 -3608.9,E2 -3608.9} C_VEL
LIN {X 0,Y 545.108,Z 316.212,A -85,B 0,C 180,E1 -3611.905,E2 -3611.905} C_VEL
LIN {X 0,Y 545.089,Z 316.205,A -85,B 0,C 180,E1 -3614.943,E2 -3614.943} C_VEL
LIN {X 0,Y 545.064,Z 316.216,A -85,B 0,C 180,E1 -3618.026,E2 -3618.026} C_VEL
LIN {X 0,Y 545.095,Z 316.208,A -85,B 0,C 180,E1 -3620.372,E2 -3620.372} C_VEL
LIN {X 0,Y 545.081,Z 316.212,A -85,B 0,C 180,E1 -3623.559,E2 -3623.559} C_VEL
LIN {X 0,Y 545.078,Z 316.214,A -85,B 0,C 180,E1 -3626.001,E2 -3626.001} C_VEL
LIN {X 0,Y 545.072,Z 316.208,A -85,B 0,C 180,E1 -3628.744,E2 -3628.744} C_VEL
LIN {X 0,Y 545.061,Z 316.219,A -85,B 0,C 180,E1 -3631.679,E2 -3631.679} C_VEL
LIN {X 0,Y 545.068,Z 316.209,A -85,B 0,C 180,E1 -3634.564,E2 -3634.564} C_VEL
LIN {X 0,Y 545.035,Z 316.218,A -85,B 0,C 180,E1 -3637.304,E2 -3637.304} C_VEL
LIN {X 0,Y 545.067,Z 316.211,A -85,B 0,C 180,E1 -3640.142,E2 -3640.142} C_VEL
LIN {X 0,Y 545.081,Z 316.211,A -85,B 0,C 180,E1 -3643.106,E2 -3643.106} C_VEL
LIN {X 0,Y 545.051,Z 316.212,A -85,B 0,C 180,E1 -3646.226,E2 -3646.226} C_VEL
LIN {X 0,Y 545.083,Z 316.209,A -85,B 0,C 180,E1 -3648.885,E2 -3648.885} C_VEL
LIN {X 0,Y 545.082,Z 316.209,A -85,B 0,C 180,E1 -3650.818,E2 -3650.818} C_VEL
LIN {X 0,Y 545.053,Z 316.219,A -85,B 0,C 180,E1 -3653.62,E2 -3653.62} C_VEL
LIN {X 0,Y 545.069,Z 316.211,A -85,B 0,C 180,E1 -3656.328,E2 -3656.328} C_VEL
LIN {X 0,Y 545.068,Z 316.213,A -85,B 0,C 180,E1 -3658.952,E2 -3658.952} C_VEL
LIN {X 0,Y 545.103,Z 316.212,A -85,B 0,C 180,E1 -3661.508,E2 -3661.508} C_VEL
LIN {X 0,Y 545.118,Z 316.245,A -85,B 0,C 180,E1 -3664.656,E2 -3664.656} C_VEL
LIN {X 0,Y 546.701,Z 324.375,A -85,B 0,C 180,E1 -3665.885,E2 -3665.885} C_VEL
LIN {X 0,Y 546.308,Z 344.561,A -85,B 0,C 180,E1 -3668.689,E2 -3668.689} C_VEL
LIN {X 0,Y 545.93,Z 365.972,A -85,B 0,C 180,E1 -3671.615,E2 -3671.615} C_VEL
LIN {X 0,Y 545.826,Z 371.442,A -85,B 0,C 180,E1 -3672.356,E2 -3672.356} C_VEL
LIN {X 0,Y 547.459,Z 380.815,A -85,B 0,C 180,E1 -3672.538,E2 -3672.538} C_VEL
LIN {X 0,Y 546.934,Z 508.599,A -85,B 0,C 180,E1 -3674.249,E2 -3674.249} C_VEL
LIN {X 0,Y 546.742,Z 522.733,A -85,B 0,C 180,E1 -3674.575,E2 -3674.575} C_VEL
LIN {X 0,Y 546.59,Z 535.737,A -85,B 0,C 180,E1 -3675.016,E2 -3675.016} C_VEL
LIN {X 0,Y 546.321,Z 548.096,A -85,B 0,C 180,E1 -3675.567,E2 -3675.567} C_VEL
LIN {X 0,Y 546.026,Z 561.245,A -85,B 0,C 180,E1 -3676.319,E2 -3676.319} C_VEL
LIN {X 0,Y 545.731,Z 573.132,A -85,B 0,C 180,E1 -3677.165,E2 -3677.165} C_VEL
LIN {X 0,Y 545.472,Z 583.985,A -85,B 0,C 180,E1 -3678.103,E2 -3678.103} C_VEL
LIN {X 0,Y 545.232,Z 594.706,A -85,B 0,C 180,E1 -3679.228,E2 -3679.228} C_VEL
LIN {X 0,Y 545.024,Z 603.556,A -85,B 0,C 180,E1 -3680.35,E2 -3680.35} C_VEL
LIN {X 0,Y 544.872,Z 612.034,A -85,B 0,C 180,E1 -3681.656,E2 -3681.656} C_VEL
LIN {X 0,Y 544.736,Z 618.863,A -85,B 0,C 180,E1 -3682.96,E2 -3682.96} C_VEL
LIN {X 0,Y 544.731,Z 623.569,A -85,B 0,C 180,E1 -3684.076,E2 -3684.076} C_VEL
LIN {X 0,Y 544.654,Z 628.444,A -85,B 0,C 180,E1 -3685.56,E2 -3685.56} C_VEL
LIN {X 0,Y 544.646,Z 631.832,A -85,B 0,C 180,E1 -3687.041,E2 -3687.041} C_VEL
LIN {X 0,Y 544.541,Z 633.834,A -85,B 0,C 180,E1 -3688.521,E2 -3688.521} C_VEL
LIN {X 0,Y 544.539,Z 634.5,A -85,B 0,C 180,E1 -3690,E2 -3690} C_VEL
LIN {X 0,Y 544.541,Z 633.836,A -85,B 0,C 180,E1 -3691.479,E2 -3691.479} C_VEL
LIN {X 0,Y 544.646,Z 631.835,A -85,B 0,C 180,E1 -3692.959,E2 -3692.959} C_VEL
LIN {X 0,Y 544.654,Z 628.447,A -85,B 0,C 180,E1 -3694.44,E2 -3694.44} C_VEL
LIN {X 0,Y 544.735,Z 623.567,A -85,B 0,C 180,E1 -3695.924,E2 -3695.924} C_VEL
LIN {X 0,Y 544.783,Z 617.054,A -85,B 0,C 180,E1 -3697.412,E2 -3697.412} C_VEL
LIN {X 0,Y 544.911,Z 609.803,A -85,B 0,C 180,E1 -3698.717,E2 -3698.717} C_VEL
LIN {X 0,Y 545.081,Z 600.821,A -85,B 0,C 180,E1 -3700.024,E2 -3700.024} C_VEL
LIN {X 0,Y 545.35,Z 591.392,A -85,B 0,C 180,E1 -3701.146,E2 -3701.146} C_VEL
LIN {X 0,Y 545.545,Z 580.95,A -85,B 0,C 180,E1 -3702.178,E2 -3702.178} C_VEL
LIN {X 0,Y 545.796,Z 569.425,A -85,B 0,C 180,E1 -3703.118,E2 -3703.118} C_VEL
LIN {X 0,Y 546.104,Z 556.635,A -85,B 0,C 180,E1 -3703.963,E2 -3703.963} C_VEL
LIN {X 0,Y 546.403,Z 544.14,A -85,B 0,C 180,E1 -3704.621,E2 -3704.621} C_VEL
LIN {X 0,Y 546.674,Z 530.193,A -85,B 0,C 180,E1 -3705.187,E2 -3705.187} C_VEL
LIN {X 0,Y 546.861,Z 516.039,A -85,B 0,C 180,E1 -3705.598,E2 -3705.598} C_VEL
LIN {X 0,Y 546.984,Z 500.775,A -85,B 0,C 180,E1 -3705.869,E2 -3705.869} C_VEL
LIN {X 0,Y 547.432,Z 380.2,A -85,B 0,C 180,E1 -3707.471,E2 -3707.471} C_VEL
LIN {X 0,Y 545.82,Z 371.245,A -85,B 0,C 180,E1 -3707.669,E2 -3707.669} C_VEL
LIN {X 0,Y 546.226,Z 350.226,A -85,B 0,C 180,E1 -3710.525,E2 -3710.525} C_VEL
LIN {X 0,Y 546.658,Z 327.686,A -85,B 0,C 180,E1 -3713.647,E2 -3713.647} C_VEL
LIN {X 0,Y 546.584,Z 323.117,A -85,B 0,C 180,E1 -3714.297,E2 -3714.297} C_VEL
LIN {X 0,Y 545.115,Z 316.211,A -85,B 0,C 180,E1 -3715.366,E2 -3715.366} C_VEL
LIN {X 0,Y 545.104,Z 316.213,A -85,B 0,C 180,E1 -3718.492,E2 -3718.492} C_VEL
LIN {X 0,Y 545.068,Z 316.213,A -85,B 0,C 180,E1 -3721.048,E2 -3721.048} C_VEL
LIN {X 0,Y 545.068,Z 316.209,A -85,B 0,C 180,E1 -3723.672,E2 -3723.672} C_VEL
LIN {X 0,Y 545.072,Z 316.213,A -85,B 0,C 180,E1 -3726.926,E2 -3726.926} C_VEL
LIN {X 0,Y 545.067,Z 316.213,A -85,B 0,C 180,E1 -3730.143,E2 -3730.143} C_VEL
LIN {X 0,Y 545.081,Z 316.208,A -85,B 0,C 180,E1 -3733.107,E2 -3733.107} C_VEL
LIN {X 0,Y 545.051,Z 316.217,A -85,B 0,C 180,E1 -3736.227,E2 -3736.227} C_VEL
LIN {X 0,Y 545.084,Z 316.21,A -85,B 0,C 180,E1 -3738.886,E2 -3738.886} C_VEL
LIN {X 0,Y 545.081,Z 316.21,A -85,B 0,C 180,E1 -3740.818,E2 -3740.818} C_VEL
LIN {X 0,Y 545.037,Z 316.213,A -85,B 0,C 180,E1 -3743.619,E2 -3743.619} C_VEL
LIN {X 0,Y 545.068,Z 316.217,A -85,B 0,C 180,E1 -3746.328,E2 -3746.328} C_VEL
LIN {X 0,Y 545.069,Z 316.21,A -85,B 0,C 180,E1 -3748.952,E2 -3748.952} C_VEL
LIN {X 0,Y 545.079,Z 316.208,A -85,B 0,C 180,E1 -3751.506,E2 -3751.506} C_VEL
LIN {X 0,Y 545.108,Z 316.205,A -85,B 0,C 180,E1 -3754.82,E2 -3754.82} C_VEL
LIN {X 0,Y 545.039,Z 316.212,A -85,B 0,C 180,E1 -3757.242,E2 -3757.242} C_VEL
LIN {X 0,Y 545.12,Z 316.207,A -85,B 0,C 180,E1 -3760.415,E2 -3760.415} C_VEL
LIN {X 0,Y 545.065,Z 316.21,A -85,B 0,C 180,E1 -3763.521,E2 -3763.521} C_VEL
LIN {X 0,Y 545.097,Z 316.211,A -85,B 0,C 180,E1 -3765.82,E2 -3765.82} C_VEL
LIN {X 0,Y 545.121,Z 316.203,A -85,B 0,C 180,E1 -3768.85,E2 -3768.85} C_VEL
LIN {X 0,Y 545.088,Z 316.212,A -85,B 0,C 180,E1 -3771.847,E2 -3771.847} C_VEL
LIN {X 0,Y 545.196,Z 316.193,A -85,B 0,C 180,E1 -3774.823,E2 -3774.823} C_VEL
LIN {X 0,Y 545.194,Z 316.198,A -85,B 0,C 180,E1 -3777.784,E2 -3777.784} C_VEL
LIN {X 0,Y 545.194,Z 316.2,A -85,B 0,C 180,E1 -3780,E2 -3780} C_VEL
LIN {X 0,Y 545.161,Z 316.196,A -85,B 0,C 180,E1 -3782.956,E2 -3782.956} C_VEL
LIN {X 0,Y 545.129,Z 316.206,A -85,B 0,C 180,E1 -3785.92,E2 -3785.92} C_VEL
LIN {X 0,Y 545.095,Z 316.206,A -85,B 0,C 180,E1 -3788.901,E2 -3788.901} C_VEL
LIN {X 0,Y 545.098,Z 316.211,A -85,B 0,C 180,E1 -3791.905,E2 -3791.905} C_VEL
LIN {X 0,Y 545.081,Z 316.208,A -85,B 0,C 180,E1 -3794.944,E2 -3794.944} C_VEL
LIN {X 0,Y 545.05,Z 316.215,A -85,B 0,C 180,E1 -3798.027,E2 -3798.027} C_VEL
LIN {X 0,Y 545.036,Z 316.211,A -85,B 0,C 180,E1 -3800.375,E2 -3800.375} C_VEL
LIN {X 0,Y 544.992,Z 316.219,A -85,B 0,C 180,E1 -3802.76,E2 -3802.76} C_VEL
LIN {X 0,Y 545.039,Z 316.219,A -85,B 0,C 180,E1 -3805.495,E2 -3805.495} C_VEL
LIN {X 0,Y 545.036,Z 316.211,A -85,B 0,C 180,E1 -3808.496,E2 -3808.496} C_VEL
LIN {X 0,Y 545.047,Z 316.217,A -85,B 0,C 180,E1 -3811.676,E2 -3811.676} C_VEL
LIN {X 0,Y 545.047,Z 316.211,A -85,B 0,C 180,E1 -3814.566,E2 -3814.566} C_VEL
LIN {X 0,Y 545.001,Z 316.215,A -85,B 0,C 180,E1 -3816.962,E2 -3816.962} C_VEL
LIN {X 0,Y 544.335,Z 316.307,A -85,B 0,C 180,E1 -3817.579,E2 -3817.579} C_VEL
LIN {X 0,Y 541.481,Z 316.661,A -85,B 0,C 180,E1 -3818.58,E2 -3818.58} C_VEL
LIN {X 0,Y 539.067,Z 316.966,A -85,B 0,C 180,E1 -3819.386,E2 -3819.386} C_VEL
LIN {X 0,Y 538.029,Z 317.087,A -85,B 0,C 180,E1 -3820.008,E2 -3820.008} C_VEL
LIN {X 0,Y 537.944,Z 317.096,A -85,B 0,C 180,E1 -3820.219,E2 -3820.219} C_VEL
LIN {X 0,Y 537.957,Z 317.099,A -85,B 0,C 180,E1 -3822.979,E2 -3822.979} C_VEL
LIN {X 0,Y 537.996,Z 317.09,A -85,B 0,C 180,E1 -3825.93,E2 -3825.93} C_VEL
LIN {X 0,Y 537.976,Z 317.094,A -85,B 0,C 180,E1 -3828.221,E2 -3828.221} C_VEL
LIN {X 0,Y 537.974,Z 317.102,A -85,B 0,C 180,E1 -3831.166,E2 -3831.166} C_VEL
LIN {X 0,Y 537.959,Z 317.096,A -85,B 0,C 180,E1 -3834.095,E2 -3834.095} C_VEL
LIN {X 0,Y 538.002,Z 317.093,A -85,B 0,C 180,E1 -3836.725,E2 -3836.725} C_VEL
LIN {X 0,Y 537.992,Z 317.097,A -85,B 0,C 180,E1 -3839.564,E2 -3839.564} C_VEL
LIN {X 0,Y 537.994,Z 317.098,A -85,B 0,C 180,E1 -3842.662,E2 -3842.662} C_VEL
LIN {X 0,Y 537.998,Z 317.138,A -85,B 0,C 180,E1 -3842.792,E2 -3842.792} C_VEL
LIN {X 0,Y 539.099,Z 323.685,A -85,B 0,C 180,E1 -3843.945,E2 -3843.945} C_VEL
LIN {X 0,Y 538.76,Z 340.648,A -85,B 0,C 180,E1 -3846.758,E2 -3846.758} C_VEL
LIN {X 0,Y 538.732,Z 343.143,A -85,B 0,C 180,E1 -3847.169,E2 -3847.169} C_VEL
LIN {X 0,Y 540.698,Z 353.789,A -85,B 0,C 180,E1 -3847.39,E2 -3847.39} C_VEL
LIN {X 0,Y 540.152,Z 479.855,A -85,B 0,C 180,E1 -3849.109,E2 -3849.109} C_VEL
LIN {X 0,Y 539.923,Z 494.51,A -85,B 0,C 180,E1 -3849.468,E2 -3849.468} C_VEL
LIN {X 0,Y 539.668,Z 507.874,A -85,B 0,C 180,E1 -3849.945,E2 -3849.945} C_VEL
LIN {X 0,Y 539.389,Z 521.455,A -85,B 0,C 180,E1 -3850.594,E2 -3850.594} C_VEL
LIN {X 0,Y 539.049,Z 534.2,A -85,B 0,C 180,E1 -3851.372,E2 -3851.372} C_VEL
LIN {X 0,Y 538.737,Z 545.64,A -85,B 0,C 180,E1 -3852.235,E2 -3852.235} C_VEL
LIN {X 0,Y 538.46,Z 555.358,A -85,B 0,C 180,E1 -3853.117,E2 -3853.117} C_VEL
LIN {X 0,Y 538.166,Z 565.999,A -85,B 0,C 180,E1 -3854.277,E2 -3854.277} C_VEL
LIN {X 0,Y 537.968,Z 574.897,A -85,B 0,C 180,E1 -3855.455,E2 -3855.455} C_VEL
LIN {X 0,Y 537.757,Z 583.115,A -85,B 0,C 180,E1 -3856.779,E2 -3856.779} C_VEL
LIN {X 0,Y 537.659,Z 588.939,A -85,B 0,C 180,E1 -3857.928,E2 -3857.928} C_VEL
LIN {X 0,Y 537.622,Z 593.686,A -85,B 0,C 180,E1 -3859.073,E2 -3859.073} C_VEL
LIN {X 0,Y 537.552,Z 598.583,A -85,B 0,C 180,E1 -3860.594,E2 -3860.594} C_VEL
LIN {X 0,Y 537.518,Z 601.224,A -85,B 0,C 180,E1 -3861.731,E2 -3861.731} C_VEL
LIN {X 0,Y 537.552,Z 603.513,A -85,B 0,C 180,E1 -3863.242,E2 -3863.242} C_VEL
LIN {X 0,Y 537.517,Z 604.444,A -85,B 0,C 180,E1 -3864.749,E2 -3864.749} C_VEL
LIN {X 0,Y 537.546,Z 604.044,A -85,B 0,C 180,E1 -3866.252,E2 -3866.252} C_VEL
LIN {X 0,Y 537.488,Z 602.316,A -85,B 0,C 180,E1 -3867.752,E2 -3867.752} C_VEL
LIN {X 0,Y 537.454,Z 599.23,A -85,B 0,C 180,E1 -3869.251,E2 -3869.251} C_VEL
LIN {X 0,Y 537.513,Z 594.698,A -85,B 0,C 180,E1 -3870.749,E2 -3870.749} C_VEL
LIN {X 0,Y 537.601,Z 588.535,A -85,B 0,C 180,E1 -3872.248,E2 -3872.248} C_VEL
LIN {X 0,Y 537.808,Z 581.68,A -85,B 0,C 180,E1 -3873.559,E2 -3873.559} C_VEL
LIN {X 0,Y 538.027,Z 573.208,A -85,B 0,C 180,E1 -3874.871,E2 -3874.871} C_VEL
LIN {X 0,Y 538.253,Z 564.424,A -85,B 0,C 180,E1 -3875.996,E2 -3875.996} C_VEL
LIN {X 0,Y 538.517,Z 554.588,A -85,B 0,C 180,E1 -3877.047,E2 -3877.047} C_VEL
LIN {X 0,Y 538.798,Z 543.111,A -85,B 0,C 180,E1 -3878.061,E2 -3878.061} C_VEL
LIN {X 0,Y 539.109,Z 531.403,A -85,B 0,C 180,E1 -3878.906,E2 -3878.906} C_VEL
LIN {X 0,Y 539.441,Z 518.488,A -85,B 0,C 180,E1 -3879.656,E2 -3879.656} C_VEL
LIN {X 0,Y 539.703,Z 504.901,A -85,B 0,C 180,E1 -3880.267,E2 -3880.267} C_VEL
LIN {X 0,Y 539.966,Z 490.526,A -85,B 0,C 180,E1 -3880.736,E2 -3880.736} C_VEL
LIN {X 0,Y 540.152,Z 476.285,A -85,B 0,C 180,E1 -3881.041,E2 -3881.041} C_VEL
LIN {X 0,Y 540.629,Z 352.87,A -85,B 0,C 180,E1 -3882.715,E2 -3882.715} C_VEL
LIN {X 0,Y 538.741,Z 343.055,A -85,B 0,C 180,E1 -3882.933,E2 -3882.933} C_VEL
LIN {X 0,Y 539.138,Z 325.187,A -85,B 0,C 180,E1 -3885.887,E2 -3885.887} C_VEL
LIN {X 0,Y 538.741,Z 320.579,A -85,B 0,C 180,E1 -3886.678,E2 -3886.678} C_VEL
LIN {X 0,Y 538.021,Z 317.095,A -85,B 0,C 180,E1 -3887.321,E2 -3887.321} C_VEL
LIN {X 0,Y 538.029,Z 317.089,A -85,B 0,C 180,E1 -3889.863,E2 -3889.863} C_VEL
LIN {X 0,Y 537.997,Z 317.098,A -85,B 0,C 180,E1 -3893.073,E2 -3893.073} C_VEL
LIN {X 0,Y 537.969,Z 317.095,A -85,B 0,C 180,E1 -3895.655,E2 -3895.655} C_VEL
LIN {X 0,Y 537.972,Z 317.094,A -85,B 0,C 180,E1 -3898.054,E2 -3898.054} C_VEL
LIN {X 0,Y 537.99,Z 317.096,A -85,B 0,C 180,E1 -3900.629,E2 -3900.629} C_VEL
LIN {X 0,Y 538.002,Z 317.092,A -85,B 0,C 180,E1 -3903.275,E2 -3903.275} C_VEL
LIN {X 0,Y 537.955,Z 317.096,A -85,B 0,C 180,E1 -3906.008,E2 -3906.008} C_VEL
LIN {X 0,Y 537.975,Z 317.1,A -85,B 0,C 180,E1 -3908.834,E2 -3908.834} C_VEL
LIN {X 0,Y 537.977,Z 317.092,A -85,B 0,C 180,E1 -3911.872,E2 -3911.872} C_VEL
LIN {X 0,Y 537.987,Z 317.096,A -85,B 0,C 180,E1 -3914.865,E2 -3914.865} C_VEL
LIN {X 0,Y 537.962,Z 317.095,A -85,B 0,C 180,E1 -3917.208,E2 -3917.208} C_VEL
LIN {X 0,Y 537.973,Z 317.099,A -85,B 0,C 180,E1 -3920.423,E2 -3920.423} C_VEL
LIN {X 0,Y 537.957,Z 317.096,A -85,B 0,C 180,E1 -3923.061,E2 -3923.061} C_VEL
LIN {X 0,Y 537.999,Z 317.09,A -85,B 0,C 180,E1 -3925.825,E2 -3925.825} C_VEL
LIN {X 0,Y 537.994,Z 317.098,A -85,B 0,C 180,E1 -3928.497,E2 -3928.497} C_VEL
LIN {X 0,Y 537.988,Z 317.091,A -85,B 0,C 180,E1 -3931.095,E2 -3931.095} C_VEL
LIN {X 0,Y 537.987,Z 317.09,A -85,B 0,C 180,E1 -3933.63,E2 -3933.63} C_VEL
LIN {X 0,Y 537.987,Z 317.096,A -85,B 0,C 180,E1 -3936.128,E2 -3936.128} C_VEL
LIN {X 0,Y 538.002,Z 317.089,A -85,B 0,C 180,E1 -3938.545,E2 -3938.545} C_VEL
LIN {X 0,Y 538.01,Z 317.086,A -85,B 0,C 180,E1 -3940.939,E2 -3940.939} C_VEL
LIN {X 0,Y 537.968,Z 317.093,A -85,B 0,C 180,E1 -3943.297,E2 -3943.297} C_VEL
LIN {X 0,Y 538.046,Z 317.084,A -85,B 0,C 180,E1 -3945.63,E2 -3945.63} C_VEL
LIN {X 0,Y 538.08,Z 317.074,A -85,B 0,C 180,E1 -3948.701,E2 -3948.701} C_VEL
LIN {X 0,Y 538.06,Z 317.082,A -85,B 0,C 180,E1 -3951.739,E2 -3951.739} C_VEL
LIN {X 0,Y 538.132,Z 317.074,A -85,B 0,C 180,E1 -3954.754,E2 -3954.754} C_VEL
LIN {X 0,Y 538.165,Z 317.072,A -85,B 0,C 180,E1 -3957.754,E2 -3957.754} C_VEL
LIN {X 0,Y 538.181,Z 317.066,A -85,B 0,C 180,E1 -3960.748,E2 -3960.748} C_VEL
LIN {X 0,Y 538.124,Z 317.074,A -85,B 0,C 180,E1 -3962.994,E2 -3962.994} C_VEL
LIN {X 0,Y 538.092,Z 317.085,A -85,B 0,C 180,E1 -3965.997,E2 -3965.997} C_VEL
LIN {X 0,Y 538.053,Z 317.082,A -85,B 0,C 180,E1 -3969.018,E2 -3969.018} C_VEL
LIN {X 0,Y 538.067,Z 317.088,A -85,B 0,C 180,E1 -3972.063,E2 -3972.063} C_VEL
LIN {X 0,Y 538.048,Z 317.083,A -85,B 0,C 180,E1 -3975.144,E2 -3975.144} C_VEL
LIN {X 0,Y 538.017,Z 317.09,A -85,B 0,C 180,E1 -3978.271,E2 -3978.271} C_VEL
LIN {X 0,Y 538.04,Z 317.085,A -85,B 0,C 180,E1 -3980.651,E2 -3980.651} C_VEL
LIN {X 0,Y 538.005,Z 317.097,A -85,B 0,C 180,E1 -3983.888,E2 -3983.888} C_VEL
LIN {X 0,Y 538.039,Z 317.086,A -85,B 0,C 180,E1 -3986.367,E2 -3986.367} C_VEL
LIN {X 0,Y 538.033,Z 317.085,A -85,B 0,C 180,E1 -3988.933,E2 -3988.933} C_VEL
LIN {X 0,Y 538.013,Z 317.094,A -85,B 0,C 180,E1 -3991.887,E2 -3991.887} C_VEL
LIN {X 0,Y 538.018,Z 317.088,A -85,B 0,C 180,E1 -3994.618,E2 -3994.618} C_VEL
LIN {X 0,Y 538.003,Z 317.093,A -85,B 0,C 180,E1 -3997.169,E2 -3997.169} C_VEL
LIN {X 0,Y 538.024,Z 317.093,A -85,B 0,C 180,E1 -3999.797,E2 -3999.797} C_VEL
LIN {X 0,Y 538.021,Z 317.088,A -85,B 0,C 180,E1 -4002.786,E2 -4002.786} C_VEL
LIN {X 0,Y 538.02,Z 317.09,A -85,B 0,C 180,E1 -4005.926,E2 -4005.926} C_VEL
LIN {X 0,Y 538.032,Z 317.086,A -85,B 0,C 180,E1 -4008.227,E2 -4008.227} C_VEL
LIN {X 0,Y 538.014,Z 317.094,A -85,B 0,C 180,E1 -4011.169,E2 -4011.169} C_VEL
LIN {X 0,Y 538.026,Z 317.089,A -85,B 0,C 180,E1 -4014.084,E2 -4014.084} C_VEL
LIN {X 0,Y 538.032,Z 317.089,A -85,B 0,C 180,E1 -4016.727,E2 -4016.727} C_VEL
LIN {X 0,Y 538.028,Z 317.093,A -85,B 0,C 180,E1 -4019.556,E2 -4019.556} C_VEL
LIN {X 0,Y 538.042,Z 317.088,A -85,B 0,C 180,E1 -4021.95,E2 -4021.95} C_VEL
LIN {X 0,Y 538.073,Z 317.225,A -85,B 0,C 180,E1 -4024.467,E2 -4024.467} C_VEL
LIN {X 0,Y 539.842,Z 326.151,A -85,B 0,C 180,E1 -4025.836,E2 -4025.836} C_VEL
LIN {X 0,Y 539.33,Z 348.668,A -85,B 0,C 180,E1 -4029.001,E2 -4029.001} C_VEL
LIN {X 0,Y 538.855,Z 371.319,A -85,B 0,C 180,E1 -4032.123,E2 -4032.123} C_VEL
LIN {X 0,Y 540.687,Z 381.707,A -85,B 0,C 180,E1 -4032.327,E2 -4032.327} C_VEL
LIN {X 0,Y 540.107,Z 508.386,A -85,B 0,C 180,E1 -4034.045,E2 -4034.045} C_VEL
LIN {X 0,Y 539.892,Z 523.14,A -85,B 0,C 180,E1 -4034.393,E2 -4034.393} C_VEL
LIN {X 0,Y 539.696,Z 535.781,A -85,B 0,C 180,E1 -4034.829,E2 -4034.829} C_VEL
LIN {X 0,Y 539.439,Z 547.945,A -85,B 0,C 180,E1 -4035.379,E2 -4035.379} C_VEL
LIN {X 0,Y 539.106,Z 561.136,A -85,B 0,C 180,E1 -4036.14,E2 -4036.14} C_VEL
LIN {X 0,Y 538.788,Z 573.068,A -85,B 0,C 180,E1 -4036.996,E2 -4036.996} C_VEL
LIN {X 0,Y 538.489,Z 583.969,A -85,B 0,C 180,E1 -4037.947,E2 -4037.947} C_VEL
LIN {X 0,Y 538.229,Z 594.705,A -85,B 0,C 180,E1 -4039.086,E2 -4039.086} C_VEL
LIN {X 0,Y 537.976,Z 603.555,A -85,B 0,C 180,E1 -4040.222,E2 -4040.222} C_VEL
LIN {X 0,Y 537.824,Z 612.033,A -85,B 0,C 180,E1 -4041.546,E2 -4041.546} C_VEL
LIN {X 0,Y 537.661,Z 618.863,A -85,B 0,C 180,E1 -4042.867,E2 -4042.867} C_VEL
LIN {X 0,Y 537.654,Z 624.96,A -85,B 0,C 180,E1 -4044.374,E2 -4044.374} C_VEL
LIN {X 0,Y 537.55,Z 628.444,A -85,B 0,C 180,E1 -4045.501,E2 -4045.501} C_VEL
LIN {X 0,Y 537.547,Z 631.832,A -85,B 0,C 180,E1 -4047.002,E2 -4047.002} C_VEL
LIN {X 0,Y 537.447,Z 633.835,A -85,B 0,C 180,E1 -4048.501,E2 -4048.501} C_VEL
LIN {X 0,Y 537.44,Z 634.5,A -85,B 0,C 180,E1 -4050,E2 -4050} C_VEL
LIN {X 0,Y 537.447,Z 633.836,A -85,B 0,C 180,E1 -4051.499,E2 -4051.499} C_VEL
LIN {X 0,Y 537.547,Z 631.836,A -85,B 0,C 180,E1 -4052.998,E2 -4052.998} C_VEL
LIN {X 0,Y 537.55,Z 628.446,A -85,B 0,C 180,E1 -4054.499,E2 -4054.499} C_VEL
LIN {X 0,Y 537.647,Z 623.567,A -85,B 0,C 180,E1 -4056.003,E2 -4056.003} C_VEL
LIN {X 0,Y 537.704,Z 617.053,A -85,B 0,C 180,E1 -4057.51,E2 -4057.51} C_VEL
LIN {X 0,Y 537.86,Z 609.803,A -85,B 0,C 180,E1 -4058.832,E2 -4058.832} C_VEL
LIN {X 0,Y 538.048,Z 600.82,A -85,B 0,C 180,E1 -4060.157,E2 -4060.157} C_VEL
LIN {X 0,Y 538.342,Z 591.391,A -85,B 0,C 180,E1 -4061.293,E2 -4061.293} C_VEL
LIN {X 0,Y 538.565,Z 580.919,A -85,B 0,C 180,E1 -4062.339,E2 -4062.339} C_VEL
LIN {X 0,Y 538.851,Z 569.344,A -85,B 0,C 180,E1 -4063.29,E2 -4063.29} C_VEL
LIN {X 0,Y 539.184,Z 556.507,A -85,B 0,C 180,E1 -4064.146,E2 -4064.146} C_VEL
LIN {X 0,Y 539.516,Z 543.973,A -85,B 0,C 180,E1 -4064.812,E2 -4064.812} C_VEL
LIN {X 0,Y 539.796,Z 530.858,A -85,B 0,C 180,E1 -4065.353,E2 -4065.353} C_VEL
LIN {X 0,Y 539.984,Z 517.204,A -85,B 0,C 180,E1 -4065.765,E2 -4065.765} C_VEL
LIN {X 0,Y 540.143,Z 502.336,A -85,B 0,C 180,E1 -4066.051,E2 -4066.051} C_VEL
LIN {X 0,Y 540.654,Z 381.345,A -85,B 0,C 180,E1 -4067.679,E2 -4067.679} C_VEL
LIN {X 0,Y 538.86,Z 371.077,A -85,B 0,C 180,E1 -4067.9,E2 -4067.9} C_VEL
LIN {X 0,Y 539.277,Z 351.459,A -85,B 0,C 180,E1 -4070.602,E2 -4070.602} C_VEL
LIN {X 0,Y 539.792,Z 330.082,A -85,B 0,C 180,E1 -4073.601,E2 -4073.601} C_VEL
LIN {X 0,Y 539.657,Z 324.543,A -85,B 0,C 180,E1 -4074.4,E2 -4074.4} C_VEL
LIN {X 0,Y 538.062,Z 317.089,A -85,B 0,C 180,E1 -4075.564,E2 -4075.564} C_VEL
LIN {X 0,Y 538.042,Z 317.089,A -85,B 0,C 180,E1 -4078.05,E2 -4078.05} C_VEL
LIN {X 0,Y 538.023,Z 317.092,A -85,B 0,C 180,E1 -4080.627,E2 -4080.627} C_VEL
LIN {X 0,Y 538.048,Z 317.085,A -85,B 0,C 180,E1 -4083.283,E2 -4083.283} C_VEL
LIN {X 0,Y 537.997,Z 317.093,A -85,B 0,C 180,E1 -4086.005,E2 -4086.005} C_VEL
LIN {X 0,Y 538.015,Z 317.092,A -85,B 0,C 180,E1 -4088.831,E2 -4088.831} C_VEL
LIN {X 0,Y 538.032,Z 317.086,A -85,B 0,C 180,E1 -4091.774,E2 -4091.774} C_VEL
LIN {X 0,Y 538.007,Z 317.092,A -85,B 0,C 180,E1 -4094.863,E2 -4094.863} C_VEL
LIN {X 0,Y 538.021,Z 317.087,A -85,B 0,C 180,E1 -4097.214,E2 -4097.214} C_VEL
LIN {X 0,Y 538.024,Z 317.093,A -85,B 0,C 180,E1 -4100.203,E2 -4100.203} C_VEL
LIN {X 0,Y 538.021,Z 317.087,A -85,B 0,C 180,E1 -4103.067,E2 -4103.067} C_VEL
LIN {X 0,Y 538.021,Z 317.089,A -85,B 0,C 180,E1 -4105.827,E2 -4105.827} C_VEL
LIN {X 0,Y 538.012,Z 317.094,A -85,B 0,C 180,E1 -4108.499,E2 -4108.499} C_VEL
LIN {X 0,Y 538.021,Z 317.087,A -85,B 0,C 180,E1 -4111.098,E2 -4111.098} C_VEL
LIN {X 0,Y 538.02,Z 317.088,A -85,B 0,C 180,E1 -4113.632,E2 -4113.632} C_VEL
LIN {X 0,Y 538.011,Z 317.096,A -85,B 0,C 180,E1 -4116.122,E2 -4116.122} C_VEL
LIN {X 0,Y 538.041,Z 317.084,A -85,B 0,C 180,E1 -4119.349,E2 -4119.349} C_VEL
LIN {X 0,Y 538.04,Z 317.087,A -85,B 0,C 180,E1 -4122.468,E2 -4122.468} C_VEL
LIN {X 0,Y 538.067,Z 317.084,A -85,B 0,C 180,E1 -4125.631,E2 -4125.631} C_VEL
LIN {X 0,Y 538.081,Z 317.08,A -85,B 0,C 180,E1 -4128.702,E2 -4128.702} C_VEL
LIN {X 0,Y 538.055,Z 317.086,A -85,B 0,C 180,E1 -4131.739,E2 -4131.739} C_VEL
LIN {X 0,Y 538.152,Z 317.071,A -85,B 0,C 180,E1 -4134.755,E2 -4134.755} C_VEL
LIN {X 0,Y 538.166,Z 317.073,A -85,B 0,C 180,E1 -4137.755,E2 -4137.755} C_VEL
LIN {X 0,Y 538.162,Z 317.076,A -85,B 0,C 180,E1 -4140,E2 -4140} C_VEL
LIN {X 0,Y 538.129,Z 317.072,A -85,B 0,C 180,E1 -4142.995,E2 -4142.995} C_VEL
LIN {X 0,Y 538.081,Z 317.083,A -85,B 0,C 180,E1 -4145.998,E2 -4145.998} C_VEL
LIN {X 0,Y 538.049,Z 317.084,A -85,B 0,C 180,E1 -4149.018,E2 -4149.018} C_VEL
LIN {X 0,Y 538.057,Z 317.086,A -85,B 0,C 180,E1 -4152.063,E2 -4152.063} C_VEL
LIN {X 0,Y 538.041,Z 317.086,A -85,B 0,C 180,E1 -4155.144,E2 -4155.144} C_VEL
LIN {X 0,Y 538.005,Z 317.09,A -85,B 0,C 180,E1 -4158.271,E2 -4158.271} C_VEL
LIN {X 0,Y 537.993,Z 317.088,A -85,B 0,C 180,E1 -4160.654,E2 -4160.654} C_VEL
LIN {X 0,Y 537.98,Z 317.094,A -85,B 0,C 180,E1 -4163.074,E2 -4163.074} C_VEL
LIN {X 0,Y 537.998,Z 317.098,A -85,B 0,C 180,E1 -4165.661,E2 -4165.661} C_VEL
LIN {X 0,Y 537.975,Z 317.093,A -85,B 0,C 180,E1 -4168.054,E2 -4168.054} C_VEL
LIN {X 0,Y 537.991,Z 317.084,A -85,B 0,C 180,E1 -4170.629,E2 -4170.629} C_VEL
LIN {X 0,Y 538.024,Z 317.092,A -85,B 0,C 180,E1 -4173.279,E2 -4173.279} C_VEL
LIN {X 0,Y 537.957,Z 317.091,A -85,B 0,C 180,E1 -4176.008,E2 -4176.008} C_VEL
LIN {X 0,Y 537.976,Z 317.094,A -85,B 0,C 180,E1 -4178.834,E2 -4178.834} C_VEL
LIN {X 0,Y 537.944,Z 317.096,A -85,B 0,C 180,E1 -4180.219,E2 -4180.219} C_VEL
LIN {X 0,Y 537.279,Z 317.181,A -85,B 0,C 180,E1 -4180.844,E2 -4180.844} C_VEL
LIN {X 0,Y 534.439,Z 317.543,A -85,B 0,C 180,E1 -4181.86,E2 -4181.86} C_VEL
LIN {X 0,Y 532.039,Z 317.846,A -85,B 0,C 180,E1 -4182.677,E2 -4182.677} C_VEL
LIN {X 0,Y 531.007,Z 317.971,A -85,B 0,C 180,E1 -4183.308,E2 -4183.308} C_VEL
LIN {X 0,Y 530.922,Z 317.978,A -85,B 0,C 180,E1 -4183.522,E2 -4183.522} C_VEL
LIN {X 0,Y 530.962,Z 317.97,A -85,B 0,C 180,E1 -4185.624,E2 -4185.624} C_VEL
LIN {X 0,Y 530.907,Z 317.975,A -85,B 0,C 180,E1 -4188.556,E2 -4188.556} C_VEL
LIN {X 0,Y 530.92,Z 317.978,A -85,B 0,C 180,E1 -4191.526,E2 -4191.526} C_VEL
LIN {X 0,Y 530.929,Z 317.972,A -85,B 0,C 180,E1 -4194.378,E2 -4194.378} C_VEL
LIN {X 0,Y 530.947,Z 317.976,A -85,B 0,C 180,E1 -4197.132,E2 -4197.132} C_VEL
LIN {X 0,Y 530.932,Z 317.974,A -85,B 0,C 180,E1 -4199.8,E2 -4199.8} C_VEL
LIN {X 0,Y 530.972,Z 318.032,A -85,B 0,C 180,E1 -4202.607,E2 -4202.607} C_VEL
LIN {X 0,Y 532.19,Z 325.251,A -85,B 0,C 180,E1 -4203.897,E2 -4203.897} C_VEL
LIN {X 0,Y 531.794,Z 342.941,A -85,B 0,C 180,E1 -4206.859,E2 -4206.859} C_VEL
LIN {X 0,Y 531.768,Z 343.39,A -85,B 0,C 180,E1 -4206.933,E2 -4206.933} C_VEL
LIN {X 0,Y 533.948,Z 354.538,A -85,B 0,C 180,E1 -4207.167,E2 -4207.167} C_VEL
LIN {X 0,Y 533.345,Z 480.299,A -85,B 0,C 180,E1 -4208.906,E2 -4208.906} C_VEL
LIN {X 0,Y 533.092,Z 494.997,A -85,B 0,C 180,E1 -4209.273,E2 -4209.273} C_VEL
LIN {X 0,Y 532.807,Z 508.733,A -85,B 0,C 180,E1 -4209.775,E2 -4209.775} C_VEL
LIN {X 0,Y 532.498,Z 522.197,A -85,B 0,C 180,E1 -4210.433,E2 -4210.433} C_VEL
LIN {X 0,Y 532.124,Z 534.836,A -85,B 0,C 180,E1 -4211.22,E2 -4211.22} C_VEL
LIN {X 0,Y 531.803,Z 546.088,A -85,B 0,C 180,E1 -4212.086,E2 -4212.086} C_VEL
LIN {X 0,Y 531.441,Z 556.845,A -85,B 0,C 180,E1 -4213.086,E2 -4213.086} C_VEL
LIN {X 0,Y 531.157,Z 567.245,A -85,B 0,C 180,E1 -4214.261,E2 -4214.261} C_VEL
LIN {X 0,Y 530.907,Z 575.793,A -85,B 0,C 180,E1 -4215.433,E2 -4215.433} C_VEL
LIN {X 0,Y 530.706,Z 583.913,A -85,B 0,C 180,E1 -4216.795,E2 -4216.795} C_VEL
LIN {X 0,Y 530.575,Z 590.42,A -85,B 0,C 180,E1 -4218.152,E2 -4218.152} C_VEL
LIN {X 0,Y 530.503,Z 596.162,A -85,B 0,C 180,E1 -4219.697,E2 -4219.697} C_VEL
LIN {X 0,Y 530.418,Z 599.417,A -85,B 0,C 180,E1 -4220.851,E2 -4220.851} C_VEL
LIN {X 0,Y 530.43,Z 602.443,A -85,B 0,C 180,E1 -4222.386,E2 -4222.386} C_VEL
LIN {X 0,Y 530.431,Z 604.103,A -85,B 0,C 180,E1 -4223.915,E2 -4223.915} C_VEL
LIN {X 0,Y 530.391,Z 604.423,A -85,B 0,C 180,E1 -4225.44,E2 -4225.44} C_VEL
LIN {X 0,Y 530.443,Z 603.415,A -85,B 0,C 180,E1 -4226.962,E2 -4226.962} C_VEL
LIN {X 0,Y 530.365,Z 601.085,A -85,B 0,C 180,E1 -4228.481,E2 -4228.481} C_VEL
LIN {X 0,Y 530.398,Z 597.382,A -85,B 0,C 180,E1 -4230,E2 -4230} C_VEL
LIN {X 0,Y 530.447,Z 592.185,A -85,B 0,C 180,E1 -4231.518,E2 -4231.518} C_VEL
LIN {X 0,Y 530.679,Z 587.155,A -85,B 0,C 180,E1 -4232.657,E2 -4232.657} C_VEL
LIN {X 0,Y 530.825,Z 580.006,A -85,B 0,C 180,E1 -4233.986,E2 -4233.986} C_VEL
LIN {X 0,Y 531.111,Z 571.18,A -85,B 0,C 180,E1 -4235.315,E2 -4235.315} C_VEL
LIN {X 0,Y 531.374,Z 561.942,A -85,B 0,C 180,E1 -4236.455,E2 -4236.455} C_VEL
LIN {X 0,Y 531.567,Z 552.542,A -85,B 0,C 180,E1 -4237.429,E2 -4237.429} C_VEL
LIN {X 0,Y 531.972,Z 540.534,A -85,B 0,C 180,E1 -4238.452,E2 -4238.452} C_VEL
LIN {X 0,Y 532.331,Z 528.145,A -85,B 0,C 180,E1 -4239.307,E2 -4239.307} C_VEL
LIN {X 0,Y 532.654,Z 516.174,A -85,B 0,C 180,E1 -4239.973,E2 -4239.973} C_VEL
LIN {X 0,Y 532.966,Z 503.021,A -85,B 0,C 180,E1 -4240.542,E2 -4240.542} C_VEL
LIN {X 0,Y 533.197,Z 488.715,A -85,B 0,C 180,E1 -4240.994,E2 -4240.994} C_VEL
LIN {X 0,Y 533.355,Z 474.677,A -85,B 0,C 180,E1 -4241.28,E2 -4241.28} C_VEL
LIN {X 0,Y 533.917,Z 354.029,A -85,B 0,C 180,E1 -4242.931,E2 -4242.931} C_VEL
LIN {X 0,Y 531.821,Z 343.356,A -85,B 0,C 180,E1 -4243.157,E2 -4243.157} C_VEL
LIN {X 0,Y 532.215,Z 325.773,A -85,B 0,C 180,E1 -4246.1,E2 -4246.1} C_VEL
LIN {X 0,Y 531.415,Z 320.137,A -85,B 0,C 180,E1 -4247.097,E2 -4247.097} C_VEL
LIN {X 0,Y 530.972,Z 317.972,A -85,B 0,C 180,E1 -4247.529,E2 -4247.529} C_VEL
LIN {X 0,Y 530.975,Z 317.968,A -85,B 0,C 180,E1 -4250.129,E2 -4250.129} C_VEL
LIN {X 0,Y 530.93,Z 317.976,A -85,B 0,C 180,E1 -4252.574,E2 -4252.574} C_VEL
LIN {X 0,Y 530.922,Z 317.98,A -85,B 0,C 180,E1 -4255.062,E2 -4255.062} C_VEL
LIN {X 0,Y 530.952,Z 317.969,A -85,B 0,C 180,E1 -4257.599,E2 -4257.599} C_VEL
LIN {X 0,Y 530.944,Z 317.973,A -85,B 0,C 180,E1 -4260.639,E2 -4260.639} C_VEL
LIN {X 0,Y 530.947,Z 317.969,A -85,B 0,C 180,E1 -4263.496,E2 -4263.496} C_VEL
LIN {X 0,Y 530.9,Z 317.975,A -85,B 0,C 180,E1 -4266.146,E2 -4266.146} C_VEL
LIN {X 0,Y 530.938,Z 317.97,A -85,B 0,C 180,E1 -4269.448,E2 -4269.448} C_VEL
LIN {X 0,Y 530.907,Z 317.978,A -85,B 0,C 180,E1 -4272.464,E2 -4272.464} C_VEL
LIN {X 0,Y 530.961,Z 317.966,A -85,B 0,C 180,E1 -4275.45,E2 -4275.45} C_VEL
LIN {X 0,Y 530.911,Z 317.98,A -85,B 0,C 180,E1 -4278.556,E2 -4278.556} C_VEL
LIN {X 0,Y 530.923,Z 317.971,A -85,B 0,C 180,E1 -4281.526,E2 -4281.526} C_VEL
LIN {X 0,Y 530.932,Z 317.976,A -85,B 0,C 180,E1 -4284.378,E2 -4284.378} C_VEL
LIN {X 0,Y 530.958,Z 317.965,A -85,B 0,C 180,E1 -4287.132,E2 -4287.132} C_VEL
LIN {X 0,Y 530.933,Z 317.971,A -85,B 0,C 180,E1 -4289.8,E2 -4289.8} C_VEL
LIN {X 0,Y 530.958,Z 317.972,A -85,B 0,C 180,E1 -4292.48,E2 -4292.48} C_VEL
LIN {X 0,Y 530.952,Z 317.969,A -85,B 0,C 180,E1 -4294.939,E2 -4294.939} C_VEL
LIN {X 0,Y 530.955,Z 317.972,A -85,B 0,C 180,E1 -4298.246,E2 -4298.246} C_VEL
LIN {X 0,Y 530.966,Z 317.966,A -85,B 0,C 180,E1 -4300.676,E2 -4300.676} C_VEL
LIN {X 0,Y 530.932,Z 317.97,A -85,B 0,C 180,E1 -4303.069,E2 -4303.069} C_VEL
LIN {X 0,Y 531.006,Z 317.96,A -85,B 0,C 180,E1 -4305.435,E2 -4305.435} C_VEL
LIN {X 0,Y 531.038,Z 317.952,A -85,B 0,C 180,E1 -4308.549,E2 -4308.549} C_VEL
LIN {X 0,Y 531.036,Z 317.956,A -85,B 0,C 180,E1 -4311.629,E2 -4311.629} C_VEL
LIN {X 0,Y 531.093,Z 317.951,A -85,B 0,C 180,E1 -4314.685,E2 -4314.685} C_VEL
LIN {X 0,Y 531.137,Z 317.947,A -85,B 0,C 180,E1 -4317.725,E2 -4317.725} C_VEL
LIN {X 0,Y 531.152,Z 317.941,A -85,B 0,C 180,E1 -4320.758,E2 -4320.758} C_VEL
LIN {X 0,Y 531.065,Z 317.953,A -85,B 0,C 180,E1 -4323.034,E2 -4323.034} C_VEL
LIN {X 0,Y 531.051,Z 317.963,A -85,B 0,C 180,E1 -4326.077,E2 -4326.077} C_VEL
LIN {X 0,Y 531.015,Z 317.959,A -85,B 0,C 180,E1 -4329.138,E2 -4329.138} C_VEL
LIN {X 0,Y 531.053,Z 317.959,A -85,B 0,C 180,E1 -4331.67,E2 -4331.67} C_VEL
LIN {X 0,Y 531.035,Z 317.956,A -85,B 0,C 180,E1 -4334.956,E2 -4334.956} C_VEL
LIN {X 0,Y 530.983,Z 317.97,A -85,B 0,C 180,E1 -4337.723,E2 -4337.723} C_VEL
LIN {X 0,Y 531.028,Z 317.963,A -85,B 0,C 180,E1 -4340.127,E2 -4340.127} C_VEL
LIN {X 0,Y 530.948,Z 317.968,A -85,B 0,C 180,E1 -4342.573,E2 -4342.573} C_VEL
LIN {X 0,Y 530.992,Z 317.963,A -85,B 0,C 180,E1 -4345.058,E2 -4345.058} C_VEL
LIN {X 0,Y 530.973,Z 317.972,A -85,B 0,C 180,E1 -4347.598,E2 -4347.598} C_VEL
LIN {X 0,Y 530.971,Z 317.968,A -85,B 0,C 180,E1 -4350.197,E2 -4350.197} C_VEL
LIN {X 0,Y 530.97,Z 317.965,A -85,B 0,C 180,E1 -4352.866,E2 -4352.866} C_VEL
LIN {X 0,Y 530.96,Z 317.975,A -85,B 0,C 180,E1 -4355.62,E2 -4355.62} C_VEL
LIN {X 0,Y 530.966,Z 317.965,A -85,B 0,C 180,E1 -4358.653,E2 -4358.653} C_VEL
LIN {X 0,Y 530.995,Z 317.97,A -85,B 0,C 180,E1 -4361.435,E2 -4361.435} C_VEL
LIN {X 0,Y 530.975,Z 317.965,A -85,B 0,C 180,E1 -4364.548,E2 -4364.548} C_VEL
LIN {X 0,Y 530.983,Z 317.968,A -85,B 0,C 180,E1 -4367.834,E2 -4367.834} C_VEL
LIN {X 0,Y 530.987,Z 317.964,A -85,B 0,C 180,E1 -4370.556,E2 -4370.556} C_VEL
LIN {X 0,Y 530.968,Z 317.975,A -85,B 0,C 180,E1 -4373.442,E2 -4373.442} C_VEL
LIN {X 0,Y 531.001,Z 317.964,A -85,B 0,C 180,E1 -4376.494,E2 -4376.494} C_VEL
LIN {X 0,Y 530.976,Z 317.973,A -85,B 0,C 180,E1 -4379.355,E2 -4379.355} C_VEL
LIN {X 0,Y 531.014,Z 317.963,A -85,B 0,C 180,E1 -4382.467,E2 -4382.467} C_VEL
LIN {X 0,Y 531.02,Z 317.973,A -85,B 0,C 180,E1 -4384.239,E2 -4384.239} C_VEL
LIN {X 0,Y 532.918,Z 327.168,A -85,B 0,C 180,E1 -4385.674,E2 -4385.674} C_VEL
LIN {X 0,Y 532.428,Z 348.464,A -85,B 0,C 180,E1 -4388.715,E2 -4388.715} C_VEL
LIN {X 0,Y 531.898,Z 371.021,A -85,B 0,C 180,E1 -4391.877,E2 -4391.877} C_VEL
LIN {X 0,Y 533.893,Z 382.699,A -85,B 0,C 180,E1 -4392.111,E2 -4392.111} C_VEL
LIN {X 0,Y 533.287,Z 509.435,A -85,B 0,C 180,E1 -4393.86,E2 -4393.86} C_VEL
LIN {X 0,Y 533.04,Z 523.579,A -85,B 0,C 180,E1 -4394.208,E2 -4394.208} C_VEL
LIN {X 0,Y 532.754,Z 537.316,A -85,B 0,C 180,E1 -4394.702,E2 -4394.702} C_VEL
LIN {X 0,Y 532.439,Z 551.29,A -85,B 0,C 180,E1 -4395.378,E2 -4395.378} C_VEL
LIN {X 0,Y 532.066,Z 563.792,A -85,B 0,C 180,E1 -4396.148,E2 -4396.148} C_VEL
LIN {X 0,Y 531.747,Z 575.221,A -85,B 0,C 180,E1 -4397.016,E2 -4397.016} C_VEL
LIN {X 0,Y 531.421,Z 586.435,A -85,B 0,C 180,E1 -4398.048,E2 -4398.048} C_VEL
LIN {X 0,Y 531.169,Z 596.177,A -85,B 0,C 180,E1 -4399.132,E2 -4399.132} C_VEL
LIN {X 0,Y 530.924,Z 604.801,A -85,B 0,C 180,E1 -4400.283,E2 -4400.283} C_VEL
LIN {X 0,Y 530.736,Z 613.062,A -85,B 0,C 180,E1 -4401.624,E2 -4401.624} C_VEL
LIN {X 0,Y 530.586,Z 618.843,A -85,B 0,C 180,E1 -4402.771,E2 -4402.771} C_VEL
LIN {X 0,Y 530.557,Z 623.569,A -85,B 0,C 180,E1 -4403.917,E2 -4403.917} C_VEL
LIN {X 0,Y 530.449,Z 628.443,A -85,B 0,C 180,E1 -4405.44,E2 -4405.44} C_VEL
LIN {X 0,Y 530.452,Z 631.832,A -85,B 0,C 180,E1 -4406.962,E2 -4406.962} C_VEL
LIN {X 0,Y 530.357,Z 633.835,A -85,B 0,C 180,E1 -4408.481,E2 -4408.481} C_VEL
LIN {X 0,Y 530.341,Z 634.5,A -85,B 0,C 180,E1 -4410,E2 -4410} C_VEL
LIN {X 0,Y 530.357,Z 633.837,A -85,B 0,C 180,E1 -4411.519,E2 -4411.519} C_VEL
LIN {X 0,Y 530.452,Z 631.836,A -85,B 0,C 180,E1 -4413.038,E2 -4413.038} C_VEL
LIN {X 0,Y 530.449,Z 628.446,A -85,B 0,C 180,E1 -4414.56,E2 -4414.56} C_VEL
LIN {X 0,Y 530.56,Z 623.567,A -85,B 0,C 180,E1 -4416.083,E2 -4416.083} C_VEL
LIN {X 0,Y 530.586,Z 618.841,A -85,B 0,C 180,E1 -4417.229,E2 -4417.229} C_VEL
LIN {X 0,Y 530.756,Z 611.969,A -85,B 0,C 180,E1 -4418.567,E2 -4418.567} C_VEL
LIN {X 0,Y 530.927,Z 603.437,A -85,B 0,C 180,E1 -4419.909,E2 -4419.909} C_VEL
LIN {X 0,Y 531.223,Z 594.539,A -85,B 0,C 180,E1 -4421.06,E2 -4421.06} C_VEL
LIN {X 0,Y 531.489,Z 583.76,A -85,B 0,C 180,E1 -4422.215,E2 -4422.215} C_VEL
LIN {X 0,Y 531.813,Z 571.678,A -85,B 0,C 180,E1 -4423.274,E2 -4423.274} C_VEL
LIN {X 0,Y 532.178,Z 559.468,A -85,B 0,C 180,E1 -4424.141,E2 -4424.141} C_VEL
LIN {X 0,Y 532.521,Z 547.727,A -85,B 0,C 180,E1 -4424.815,E2 -4424.815} C_VEL
LIN {X 0,Y 532.861,Z 534.143,A -85,B 0,C 180,E1 -4425.426,E2 -4425.426} C_VEL
LIN {X 0,Y 533.066,Z 519.954,A -85,B 0,C 180,E1 -4425.896,E2 -4425.896} C_VEL
LIN {X 0,Y 533.286,Z 505.143,A -85,B 0,C 180,E1 -4426.214,E2 -4426.214} C_VEL
LIN {X 0,Y 533.874,Z 382.318,A -85,B 0,C 180,E1 -4427.895,E2 -4427.895} C_VEL
LIN {X 0,Y 531.897,Z 370.988,A -85,B 0,C 180,E1 -4428.126,E2 -4428.126} C_VEL
LIN {X 0,Y 532.323,Z 351.269,A -85,B 0,C 180,E1 -4430.884,E2 -4430.884} C_VEL
LIN {X 0,Y 532.914,Z 331.328,A -85,B 0,C 180,E1 -4433.718,E2 -4433.718} C_VEL
LIN {X 0,Y 532.784,Z 326.186,A -85,B 0,C 180,E1 -4434.469,E2 -4434.469} C_VEL
LIN {X 0,Y 531.021,Z 317.967,A -85,B 0,C 180,E1 -4435.762,E2 -4435.762} C_VEL
LIN {X 0,Y 530.999,Z 317.969,A -85,B 0,C 180,E1 -4438.456,E2 -4438.456} C_VEL
LIN {X 0,Y 530.959,Z 317.97,A -85,B 0,C 180,E1 -4441.079,E2 -4441.079} C_VEL
LIN {X 0,Y 530.989,Z 317.963,A -85,B 0,C 180,E1 -4443.773,E2 -4443.773} C_VEL
LIN {X 0,Y 530.957,Z 317.975,A -85,B 0,C 180,E1 -4446.559,E2 -4446.559} C_VEL
LIN {X 0,Y 530.988,Z 317.963,A -85,B 0,C 180,E1 -4449.444,E2 -4449.444} C_VEL
LIN {X 0,Y 530.98,Z 317.973,A -85,B 0,C 180,E1 -4452.457,E2 -4452.457} C_VEL
LIN {X 0,Y 530.978,Z 317.964,A -85,B 0,C 180,E1 -4455.622,E2 -4455.622} C_VEL
LIN {X 0,Y 530.996,Z 317.969,A -85,B 0,C 180,E1 -4458.565,E2 -4458.565} C_VEL
LIN {X 0,Y 530.956,Z 317.966,A -85,B 0,C 180,E1 -4461.529,E2 -4461.529} C_VEL
LIN {X 0,Y 530.953,Z 317.975,A -85,B 0,C 180,E1 -4464.38,E2 -4464.38} C_VEL
LIN {X 0,Y 530.97,Z 317.965,A -85,B 0,C 180,E1 -4467.134,E2 -4467.134} C_VEL
LIN {X 0,Y 530.972,Z 317.967,A -85,B 0,C 180,E1 -4469.803,E2 -4469.803} C_VEL
LIN {X 0,Y 530.97,Z 317.97,A -85,B 0,C 180,E1 -4472.478,E2 -4472.478} C_VEL
LIN {X 0,Y 530.99,Z 317.963,A -85,B 0,C 180,E1 -4474.942,E2 -4474.942} C_VEL
LIN {X 0,Y 530.975,Z 317.971,A -85,B 0,C 180,E1 -4478.247,E2 -4478.247} C_VEL
LIN {X 0,Y 530.987,Z 317.964,A -85,B 0,C 180,E1 -4480.677,E2 -4480.677} C_VEL
LIN {X 0,Y 530.972,Z 317.964,A -85,B 0,C 180,E1 -4483.071,E2 -4483.071} C_VEL
LIN {X 0,Y 531.023,Z 317.96,A -85,B 0,C 180,E1 -4485.436,E2 -4485.436} C_VEL
LIN {X 0,Y 531.039,Z 317.959,A -85,B 0,C 180,E1 -4488.55,E2 -4488.55} C_VEL
LIN {X 0,Y 531.033,Z 317.96,A -85,B 0,C 180,E1 -4491.629,E2 -4491.629} C_VEL
LIN {X 0,Y 531.11,Z 317.948,A -85,B 0,C 180,E1 -4494.685,E2 -4494.685} C_VEL
LIN {X 0,Y 531.138,Z 317.948,A -85,B 0,C 180,E1 -4497.725,E2 -4497.725} C_VEL
LIN {X 0,Y 531.131,Z 317.951,A -85,B 0,C 180,E1 -4500,E2 -4500} C_VEL
LIN {X 0,Y 531.097,Z 317.948,A -85,B 0,C 180,E1 -4503.034,E2 -4503.034} C_VEL
LIN {X 0,Y 531.04,Z 317.958,A -85,B 0,C 180,E1 -4506.078,E2 -4506.078} C_VEL
LIN {X 0,Y 531.012,Z 317.961,A -85,B 0,C 180,E1 -4509.139,E2 -4509.139} C_VEL
LIN {X 0,Y 531.054,Z 317.961,A -85,B 0,C 180,E1 -4511.67,E2 -4511.67} C_VEL
LIN {X 0,Y 531.025,Z 317.959,A -85,B 0,C 180,E1 -4514.951,E2 -4514.951} C_VEL
LIN {X 0,Y 530.967,Z 317.966,A -85,B 0,C 180,E1 -4518.522,E2 -4518.522} C_VEL
LIN {X 0,Y 530.944,Z 317.967,A -85,B 0,C 180,E1 -4520.941,E2 -4520.941} C_VEL
LIN {X 0,Y 530.956,Z 317.968,A -85,B 0,C 180,E1 -4524.031,E2 -4524.031} C_VEL
LIN {X 0,Y 530.95,Z 317.968,A -85,B 0,C 180,E1 -4526.747,E2 -4526.747} C_VEL
LIN {X 0,Y 530.919,Z 317.976,A -85,B 0,C 180,E1 -4529.327,E2 -4529.327} C_VEL
LIN {X 0,Y 530.956,Z 317.968,A -85,B 0,C 180,E1 -4532.098,E2 -4532.098} C_VEL
LIN {X 0,Y 530.959,Z 317.968,A -85,B 0,C 180,E1 -4534.849,E2 -4534.849} C_VEL
LIN {X 0,Y 530.926,Z 317.976,A -85,B 0,C 180,E1 -4537.511,E2 -4537.511} C_VEL
LIN {X 0,Y 530.908,Z 317.972,A -85,B 0,C 180,E1 -4540.44,E2 -4540.44} C_VEL
LIN {X 0,Y 530.922,Z 317.978,A -85,B 0,C 180,E1 -4543.522,E2 -4543.522} C_VEL
LIN {X 0,Y 530.258,Z 318.057,A -85,B 0,C 180,E1 -4544.155,E2 -4544.155} C_VEL
LIN {X 0,Y 527.419,Z 318.415,A -85,B 0,C 180,E1 -4545.184,E2 -4545.184} C_VEL
LIN {X 0,Y 525.011,Z 318.712,A -85,B 0,C 180,E1 -4546.013,E2 -4546.013} C_VEL
LIN {X 0,Y 523.964,Z 318.84,A -85,B 0,C 180,E1 -4546.652,E2 -4546.652} C_VEL
LIN {X 0,Y 523.872,Z 318.851,A -85,B 0,C 180,E1 -4546.869,E2 -4546.869} C_VEL
LIN {X 0,Y 523.866,Z 318.853,A -85,B 0,C 180,E1 -4549.913,E2 -4549.913} C_VEL
LIN {X 0,Y 523.851,Z 318.858,A -85,B 0,C 180,E1 -4552.863,E2 -4552.863} C_VEL
LIN {X 0,Y 523.904,Z 318.848,A -85,B 0,C 180,E1 -4555.707,E2 -4555.707} C_VEL
LIN {X 0,Y 523.907,Z 318.847,A -85,B 0,C 180,E1 -4558.455,E2 -4558.455} C_VEL
LIN {X 0,Y 523.875,Z 318.858,A -85,B 0,C 180,E1 -4561.121,E2 -4561.121} C_VEL
LIN {X 0,Y 523.934,Z 318.892,A -85,B 0,C 180,E1 -4562.409,E2 -4562.409} C_VEL
LIN {X 0,Y 525.288,Z 326.55,A -85,B 0,C 180,E1 -4563.799,E2 -4563.799} C_VEL
LIN {X 0,Y 524.857,Z 343.551,A -85,B 0,C 180,E1 -4566.678,E2 -4566.678} C_VEL
LIN {X 0,Y 527.109,Z 354.604,A -85,B 0,C 180,E1 -4566.925,E2 -4566.925} C_VEL
LIN {X 0,Y 526.543,Z 479.49,A -85,B 0,C 180,E1 -4568.671,E2 -4568.671} C_VEL
LIN {X 0,Y 526.3,Z 494.217,A -85,B 0,C 180,E1 -4569.032,E2 -4569.032} C_VEL
LIN {X 0,Y 525.993,Z 508.048,A -85,B 0,C 180,E1 -4569.533,E2 -4569.533} C_VEL
LIN {X 0,Y 525.674,Z 521.141,A -85,B 0,C 180,E1 -4570.169,E2 -4570.169} C_VEL
LIN {X 0,Y 525.261,Z 534.023,A -85,B 0,C 180,E1 -4570.965,E2 -4570.965} C_VEL
LIN {X 0,Y 524.908,Z 545.214,A -85,B 0,C 180,E1 -4571.822,E2 -4571.822} C_VEL
LIN {X 0,Y 524.498,Z 556.354,A -85,B 0,C 180,E1 -4572.855,E2 -4572.855} C_VEL
LIN {X 0,Y 524.192,Z 566.898,A -85,B 0,C 180,E1 -4574.047,E2 -4574.047} C_VEL
LIN {X 0,Y 523.898,Z 575.545,A -85,B 0,C 180,E1 -4575.233,E2 -4575.233} C_VEL
LIN {X 0,Y 523.658,Z 583.76,A -85,B 0,C 180,E1 -4576.614,E2 -4576.614} C_VEL
LIN {X 0,Y 523.528,Z 590.339,A -85,B 0,C 180,E1 -4577.99,E2 -4577.99} C_VEL
LIN {X 0,Y 523.443,Z 594.883,A -85,B 0,C 180,E1 -4579.166,E2 -4579.166} C_VEL
LIN {X 0,Y 523.338,Z 599.464,A -85,B 0,C 180,E1 -4580.726,E2 -4580.726} C_VEL
LIN {X 0,Y 523.334,Z 602.548,A -85,B 0,C 180,E1 -4582.282,E2 -4582.282} C_VEL
LIN {X 0,Y 523.35,Z 604.25,A -85,B 0,C 180,E1 -4583.833,E2 -4583.833} C_VEL
LIN {X 0,Y 523.299,Z 604.625,A -85,B 0,C 180,E1 -4585.378,E2 -4585.378} C_VEL
LIN {X 0,Y 523.352,Z 603.678,A -85,B 0,C 180,E1 -4586.921,E2 -4586.921} C_VEL
LIN {X 0,Y 523.278,Z 601.411,A -85,B 0,C 180,E1 -4588.461,E2 -4588.461} C_VEL
LIN {X 0,Y 523.31,Z 597.766,A -85,B 0,C 180,E1 -4590,E2 -4590} C_VEL
LIN {X 0,Y 523.365,Z 592.644,A -85,B 0,C 180,E1 -4591.539,E2 -4591.539} C_VEL
LIN {X 0,Y 523.617,Z 587.667,A -85,B 0,C 180,E1 -4592.693,E2 -4592.693} C_VEL
LIN {X 0,Y 523.774,Z 580.591,A -85,B 0,C 180,E1 -4594.04,E2 -4594.04} C_VEL
LIN {X 0,Y 524.089,Z 571.86,A -85,B 0,C 180,E1 -4595.386,E2 -4595.386} C_VEL
LIN {X 0,Y 524.363,Z 562.735,A -85,B 0,C 180,E1 -4596.542,E2 -4596.542} C_VEL
LIN {X 0,Y 524.588,Z 553.506,A -85,B 0,C 180,E1 -4597.52,E2 -4597.52} C_VEL
LIN {X 0,Y 524.999,Z 542.806,A -85,B 0,C 180,E1 -4598.468,E2 -4598.468} C_VEL
LIN {X 0,Y 525.354,Z 530.947,A -85,B 0,C 180,E1 -4599.335,E2 -4599.335} C_VEL
LIN {X 0,Y 525.751,Z 517.733,A -85,B 0,C 180,E1 -4600.105,E2 -4600.105} C_VEL
LIN {X 0,Y 526.069,Z 505.005,A -85,B 0,C 180,E1 -4600.682,E2 -4600.682} C_VEL
LIN {X 0,Y 526.35,Z 490.518,A -85,B 0,C 180,E1 -4601.164,E2 -4601.164} C_VEL
LIN {X 0,Y 526.547,Z 476.023,A -85,B 0,C 180,E1 -4601.476,E2 -4601.476} C_VEL
LIN {X 0,Y 527.138,Z 354.672,A -85,B 0,C 180,E1 -4603.162,E2 -4603.162} C_VEL
LIN {X 0,Y 524.869,Z 343.455,A -85,B 0,C 180,E1 -4603.424,E2 -4603.424} C_VEL
LIN {X 0,Y 525.294,Z 326.36,A -85,B 0,C 180,E1 -4606.318,E2 -4606.318} C_VEL
LIN {X 0,Y 523.948,Z 318.846,A -85,B 0,C 180,E1 -4607.684,E2 -4607.684} C_VEL
LIN {X 0,Y 523.925,Z 318.849,A -85,B 0,C 180,E1 -4610.412,E2 -4610.412} C_VEL
LIN {X 0,Y 523.9,Z 318.855,A -85,B 0,C 180,E1 -4612.894,E2 -4612.894} C_VEL
LIN {X 0,Y 523.867,Z 318.854,A -85,B 0,C 180,E1 -4615.423,E2 -4615.423} C_VEL
LIN {X 0,Y 523.898,Z 318.848,A -85,B 0,C 180,E1 -4618.003,E2 -4618.003} C_VEL
LIN {X 0,Y 523.9,Z 318.853,A -85,B 0,C 180,E1 -4620.845,E2 -4620.845} C_VEL
LIN {X 0,Y 523.91,Z 318.845,A -85,B 0,C 180,E1 -4623.725,E2 -4623.725} C_VEL
LIN {X 0,Y 523.858,Z 318.855,A -85,B 0,C 180,E1 -4626.394,E2 -4626.394} C_VEL
LIN {X 0,Y 523.89,Z 318.851,A -85,B 0,C 180,E1 -4629.088,E2 -4629.088} C_VEL
LIN {X 0,Y 523.889,Z 318.848,A -85,B 0,C 180,E1 -4632.126,E2 -4632.126} C_VEL
LIN {X 0,Y 523.932,Z 318.842,A -85,B 0,C 180,E1 -4635.312,E2 -4635.312} C_VEL
LIN {X 0,Y 523.88,Z 318.855,A -85,B 0,C 180,E1 -4638.7,E2 -4638.7} C_VEL
LIN {X 0,Y 523.885,Z 318.848,A -85,B 0,C 180,E1 -4641.895,E2 -4641.895} C_VEL
LIN {X 0,Y 523.917,Z 318.847,A -85,B 0,C 180,E1 -4644.913,E2 -4644.913} C_VEL
LIN {X 0,Y 523.905,Z 318.843,A -85,B 0,C 180,E1 -4647.686,E2 -4647.686} C_VEL
LIN {X 0,Y 523.883,Z 318.852,A -85,B 0,C 180,E1 -4650.691,E2 -4650.691} C_VEL
LIN {X 0,Y 523.897,Z 318.848,A -85,B 0,C 180,E1 -4652.864,E2 -4652.864} C_VEL
LIN {X 0,Y 523.935,Z 318.843,A -85,B 0,C 180,E1 -4655.804,E2 -4655.804} C_VEL
LIN {X 0,Y 523.927,Z 318.838,A -85,B 0,C 180,E1 -4658.765,E2 -4658.765} C_VEL
LIN {X 0,Y 523.929,Z 318.838,A -85,B 0,C 180,E1 -4661.22,E2 -4661.22} C_VEL
LIN {X 0,Y 523.915,Z 318.85,A -85,B 0,C 180,E1 -4664.437,E2 -4664.437} C_VEL
LIN {X 0,Y 523.955,Z 318.836,A -85,B 0,C 180,E1 -4667.607,E2 -4667.607} C_VEL
LIN {X 0,Y 523.936,Z 318.837,A -85,B 0,C 180,E1 -4669.957,E2 -4669.957} C_VEL
LIN {X 0,Y 523.98,Z 318.843,A -85,B 0,C 180,E1 -4672.292,E2 -4672.292} C_VEL
LIN {X 0,Y 524.04,Z 318.831,A -85,B 0,C 180,E1 -4674.613,E2 -4674.613} C_VEL
LIN {X 0,Y 524.11,Z 318.822,A -85,B 0,C 180,E1 -4677.694,E2 -4677.694} C_VEL
LIN {X 0,Y 524.122,Z 318.817,A -85,B 0,C 180,E1 -4680.768,E2 -4680.768} C_VEL
LIN {X 0,Y 524.007,Z 318.832,A -85,B 0,C 180,E1 -4683.075,E2 -4683.075} C_VEL
LIN {X 0,Y 524.07,Z 318.825,A -85,B 0,C 180,E1 -4685.386,E2 -4685.386} C_VEL
LIN {X 0,Y 523.986,Z 318.837,A -85,B 0,C 180,E1 -4688.484,E2 -4688.484} C_VEL
LIN {X 0,Y 524.003,Z 318.838,A -85,B 0,C 180,E1 -4691.737,E2 -4691.737} C_VEL
LIN {X 0,Y 523.997,Z 318.833,A -85,B 0,C 180,E1 -4695.052,E2 -4695.052} C_VEL
LIN {X 0,Y 523.948,Z 318.846,A -85,B 0,C 180,E1 -4697.969,E2 -4697.969} C_VEL
LIN {X 0,Y 523.975,Z 318.838,A -85,B 0,C 180,E1 -4700.41,E2 -4700.41} C_VEL
LIN {X 0,Y 523.913,Z 318.844,A -85,B 0,C 180,E1 -4702.893,E2 -4702.893} C_VEL
LIN {X 0,Y 523.985,Z 318.841,A -85,B 0,C 180,E1 -4706.019,E2 -4706.019} C_VEL
LIN {X 0,Y 523.956,Z 318.842,A -85,B 0,C 180,E1 -4709.323,E2 -4709.323} C_VEL
LIN {X 0,Y 523.938,Z 318.842,A -85,B 0,C 180,E1 -4712.32,E2 -4712.32} C_VEL
LIN {X 0,Y 523.925,Z 318.847,A -85,B 0,C 180,E1 -4715.226,E2 -4715.226} C_VEL
LIN {X 0,Y 523.916,Z 318.846,A -85,B 0,C 180,E1 -4718.102,E2 -4718.102} C_VEL
LIN {X 0,Y 523.941,Z 318.844,A -85,B 0,C 180,E1 -4721.092,E2 -4721.092} C_VEL
LIN {X 0,Y 523.933,Z 318.843,A -85,B 0,C 180,E1 -4724.229,E2 -4724.229} C_VEL
LIN {X 0,Y 523.918,Z 318.845,A -85,B 0,C 180,E1 -4726.832,E2 -4726.832} C_VEL
LIN {X 0,Y 523.94,Z 318.843,A -85,B 0,C 180,E1 -4728.907,E2 -4728.907} C_VEL
LIN {X 0,Y 523.918,Z 318.849,A -85,B 0,C 180,E1 -4731.898,E2 -4731.898} C_VEL
LIN {X 0,Y 523.937,Z 318.846,A -85,B 0,C 180,E1 -4734.909,E2 -4734.909} C_VEL
LIN {X 0,Y 523.937,Z 318.848,A -85,B 0,C 180,E1 -4737.68,E2 -4737.68} C_VEL
LIN {X 0,Y 523.956,Z 318.842,A -85,B 0,C 180,E1 -4740.676,E2 -4740.676} C_VEL
LIN {X 0,Y 523.975,Z 318.844,A -85,B 0,C 180,E1 -4743.728,E2 -4743.728} C_VEL
LIN {X 0,Y 524.002,Z 318.941,A -85,B 0,C 180,E1 -4744.044,E2 -4744.044} C_VEL
LIN {X 0,Y 525.969,Z 328.33,A -85,B 0,C 180,E1 -4745.529,E2 -4745.529} C_VEL
LIN {X 0,Y 525.657,Z 342.893,A -85,B 0,C 180,E1 -4747.647,E2 -4747.647} C_VEL
LIN {X 0,Y 525.171,Z 361.087,A -85,B 0,C 180,E1 -4750.251,E2 -4750.251} C_VEL
LIN {X 0,Y 524.94,Z 370.831,A -85,B 0,C 180,E1 -4751.63,E2 -4751.63} C_VEL
LIN {X 0,Y 527.117,Z 383.588,A -85,B 0,C 180,E1 -4751.888,E2 -4751.888} C_VEL
LIN {X 0,Y 526.455,Z 509.225,A -85,B 0,C 180,E1 -4753.645,E2 -4753.645} C_VEL
LIN {X 0,Y 526.192,Z 523.895,A -85,B 0,C 180,E1 -4754.014,E2 -4754.014} C_VEL
LIN {X 0,Y 525.849,Z 538.242,A -85,B 0,C 180,E1 -4754.546,E2 -4754.546} C_VEL
LIN {X 0,Y 525.537,Z 551.085,A -85,B 0,C 180,E1 -4755.181,E2 -4755.181} C_VEL
LIN {X 0,Y 525.137,Z 563.588,A -85,B 0,C 180,E1 -4755.962,E2 -4755.962} C_VEL
LIN {X 0,Y 524.744,Z 576.194,A -85,B 0,C 180,E1 -4756.938,E2 -4756.938} C_VEL
LIN {X 0,Y 524.41,Z 586.93,A -85,B 0,C 180,E1 -4757.957,E2 -4757.957} C_VEL
LIN {X 0,Y 524.105,Z 597.502,A -85,B 0,C 180,E1 -4759.179,E2 -4759.179} C_VEL
LIN {X 0,Y 523.854,Z 605.871,A -85,B 0,C 180,E1 -4760.346,E2 -4760.346} C_VEL
LIN {X 0,Y 523.634,Z 613.873,A -85,B 0,C 180,E1 -4761.704,E2 -4761.704} C_VEL
LIN {X 0,Y 523.494,Z 620.318,A -85,B 0,C 180,E1 -4763.06,E2 -4763.06} C_VEL
LIN {X 0,Y 523.451,Z 626.033,A -85,B 0,C 180,E1 -4764.607,E2 -4764.607} C_VEL
LIN {X 0,Y 523.419,Z 630.179,A -85,B 0,C 180,E1 -4766.151,E2 -4766.151} C_VEL
LIN {X 0,Y 523.333,Z 632.885,A -85,B 0,C 180,E1 -4767.691,E2 -4767.691} C_VEL
LIN {X 0,Y 523.247,Z 634.225,A -85,B 0,C 180,E1 -4769.23,E2 -4769.23} C_VEL
LIN {X 0,Y 523.247,Z 634.226,A -85,B 0,C 180,E1 -4770.77,E2 -4770.77} C_VEL
LIN {X 0,Y 523.333,Z 632.888,A -85,B 0,C 180,E1 -4772.309,E2 -4772.309} C_VEL
LIN {X 0,Y 523.419,Z 630.183,A -85,B 0,C 180,E1 -4773.85,E2 -4773.85} C_VEL
LIN {X 0,Y 523.452,Z 626.032,A -85,B 0,C 180,E1 -4775.393,E2 -4775.393} C_VEL
LIN {X 0,Y 523.494,Z 620.314,A -85,B 0,C 180,E1 -4776.94,E2 -4776.94} C_VEL
LIN {X 0,Y 523.635,Z 613.87,A -85,B 0,C 180,E1 -4778.296,E2 -4778.296} C_VEL
LIN {X 0,Y 523.854,Z 605.866,A -85,B 0,C 180,E1 -4779.654,E2 -4779.654} C_VEL
LIN {X 0,Y 524.106,Z 597.495,A -85,B 0,C 180,E1 -4780.821,E2 -4780.821} C_VEL
LIN {X 0,Y 524.436,Z 586.753,A -85,B 0,C 180,E1 -4782.06,E2 -4782.06} C_VEL
LIN {X 0,Y 524.744,Z 576.182,A -85,B 0,C 180,E1 -4783.062,E2 -4783.062} C_VEL
LIN {X 0,Y 525.137,Z 563.578,A -85,B 0,C 180,E1 -4784.038,E2 -4784.038} C_VEL
LIN {X 0,Y 525.55,Z 551.071,A -85,B 0,C 180,E1 -4784.818,E2 -4784.818} C_VEL
LIN {X 0,Y 525.887,Z 538.216,A -85,B 0,C 180,E1 -4785.453,E2 -4785.453} C_VEL
LIN {X 0,Y 526.186,Z 523.994,A -85,B 0,C 180,E1 -4785.982,E2 -4785.982} C_VEL
LIN {X 0,Y 526.427,Z 510.343,A -85,B 0,C 180,E1 -4786.332,E2 -4786.332} C_VEL
LIN {X 0,Y 526.6,Z 482.208,A -85,B 0,C 180,E1 -4786.75,E2 -4786.75} C_VEL
LIN {X 0,Y 527.141,Z 383.494,A -85,B 0,C 180,E1 -4788.112,E2 -4788.112} C_VEL
LIN {X 0,Y 524.923,Z 370.682,A -85,B 0,C 180,E1 -4788.389,E2 -4788.389} C_VEL
LIN {X 0,Y 525.54,Z 348.24,A -85,B 0,C 180,E1 -4791.577,E2 -4791.577} C_VEL
LIN {X 0,Y 526.058,Z 329.722,A -85,B 0,C 180,E1 -4794.256,E2 -4794.256} C_VEL
LIN {X 0,Y 524.797,Z 322.575,A -85,B 0,C 180,E1 -4795.375,E2 -4795.375} C_VEL
LIN {X 0,Y 523.964,Z 318.847,A -85,B 0,C 180,E1 -4795.979,E2 -4795.979} C_VEL
LIN {X 0,Y 523.941,Z 318.847,A -85,B 0,C 180,E1 -4798.875,E2 -4798.875} C_VEL
LIN {X 0,Y 523.923,Z 318.844,A -85,B 0,C 180,E1 -4801.544,E2 -4801.544} C_VEL
LIN {X 0,Y 523.935,Z 318.846,A -85,B 0,C 180,E1 -4804.29,E2 -4804.29} C_VEL
LIN {X 0,Y 523.909,Z 318.847,A -85,B 0,C 180,E1 -4807.132,E2 -4807.132} C_VEL
LIN {X 0,Y 523.94,Z 318.844,A -85,B 0,C 180,E1 -4810.13,E2 -4810.13} C_VEL
LIN {X 0,Y 523.937,Z 318.85,A -85,B 0,C 180,E1 -4812.459,E2 -4812.459} C_VEL
LIN {X 0,Y 523.944,Z 318.84,A -85,B 0,C 180,E1 -4815.31,E2 -4815.31} C_VEL
LIN {X 0,Y 523.958,Z 318.844,A -85,B 0,C 180,E1 -4818.69,E2 -4818.69} C_VEL
LIN {X 0,Y 523.918,Z 318.844,A -85,B 0,C 180,E1 -4821.081,E2 -4821.081} C_VEL
LIN {X 0,Y 523.898,Z 318.847,A -85,B 0,C 180,E1 -4823.825,E2 -4823.825} C_VEL
LIN {X 0,Y 523.944,Z 318.844,A -85,B 0,C 180,E1 -4826.636,E2 -4826.636} C_VEL
LIN {X 0,Y 523.959,Z 318.838,A -85,B 0,C 180,E1 -4829.356,E2 -4829.356} C_VEL
LIN {X 0,Y 523.944,Z 318.848,A -85,B 0,C 180,E1 -4832.289,E2 -4832.289} C_VEL
LIN {X 0,Y 523.925,Z 318.843,A -85,B 0,C 180,E1 -4835.428,E2 -4835.428} C_VEL
LIN {X 0,Y 523.949,Z 318.841,A -85,B 0,C 180,E1 -4838.767,E2 -4838.767} C_VEL
LIN {X 0,Y 523.942,Z 318.84,A -85,B 0,C 180,E1 -4841.221,E2 -4841.221} C_VEL
LIN {X 0,Y 523.93,Z 318.844,A -85,B 0,C 180,E1 -4843.639,E2 -4843.639} C_VEL
LIN {X 0,Y 523.939,Z 318.848,A -85,B 0,C 180,E1 -4846.028,E2 -4846.028} C_VEL
LIN {X 0,Y 523.996,Z 318.834,A -85,B 0,C 180,E1 -4849.177,E2 -4849.177} C_VEL
LIN {X 0,Y 523.963,Z 318.842,A -85,B 0,C 180,E1 -4852.292,E2 -4852.292} C_VEL
LIN {X 0,Y 524.07,Z 318.826,A -85,B 0,C 180,E1 -4854.614,E2 -4854.614} C_VEL
LIN {X 0,Y 524.108,Z 318.822,A -85,B 0,C 180,E1 -4857.695,E2 -4857.695} C_VEL
LIN {X 0,Y 524.1,Z 318.827,A -85,B 0,C 180,E1 -4860,E2 -4860} C_VEL
